LIN {X 0,Y 418.26,Z 256.009,A -85,B 0,C 180,E1 -10305.113,E2 -10305.113} C_VEL
LIN {X 0,Y 418.269,Z 256.008,A -85,B 0,C 180,E1 -10308.419,E2 -10308.419} C_VEL
LIN {X 0,Y 418.275,Z 256.076,A -85,B 0,C 180,E1 -10308.94,E2 -10308.94} C_VEL
LIN {X 0,Y 420.863,Z 267.45,A -85,B 0,C 180,E1 -10311.704,E2 -10311.704} C_VEL
LIN {X 0,Y 421.563,Z 270.846,A -85,B 0,C 180,E1 -10312.505,E2 -10312.505} C_VEL
LIN {X 0,Y 424.681,Z 279.122,A -85,B 0,C 180,E1 -10312.884,E2 -10312.884} C_VEL
LIN {X 0,Y 428.293,Z 295.182,A -85,B 0,C 180,E1 -10313.417,E2 -10313.417} C_VEL
LIN {X 0,Y 426.388,Z 407.598,A -85,B 0,C 180,E1 -10315.38,E2 -10315.38} C_VEL
LIN {X 0,Y 425.814,Z 421.951,A -85,B 0,C 180,E1 -10315.821,E2 -10315.821} C_VEL
LIN {X 0,Y 425.057,Z 435.648,A -85,B 0,C 180,E1 -10316.437,E2 -10316.437} C_VEL
LIN {X 0,Y 424.136,Z 449.482,A -85,B 0,C 180,E1 -10317.277,E2 -10317.277} C_VEL
LIN {X 0,Y 423.118,Z 462.711,A -85,B 0,C 180,E1 -10318.313,E2 -10318.313} C_VEL
LIN {X 0,Y 421.977,Z 474.603,A -85,B 0,C 180,E1 -10319.472,E2 -10319.472} C_VEL
LIN {X 0,Y 420.938,Z 485.519,A -85,B 0,C 180,E1 -10320.784,E2 -10320.784} C_VEL
LIN {X 0,Y 420.063,Z 494.402,A -85,B 0,C 180,E1 -10322.066,E2 -10322.066} C_VEL
LIN {X 0,Y 419.198,Z 503.344,A -85,B 0,C 180,E1 -10323.623,E2 -10323.623} C_VEL
LIN {X 0,Y 418.524,Z 510.7,A -85,B 0,C 180,E1 -10325.178,E2 -10325.178} C_VEL
LIN {X 0,Y 417.991,Z 516.714,A -85,B 0,C 180,E1 -10326.727,E2 -10326.727} C_VEL
LIN {X 0,Y 417.581,Z 521.545,A -85,B 0,C 180,E1 -10328.269,E2 -10328.269} C_VEL
LIN {X 0,Y 417.325,Z 525.36,A -85,B 0,C 180,E1 -10329.805,E2 -10329.805} C_VEL
LIN {X 0,Y 417.115,Z 528.26,A -85,B 0,C 180,E1 -10331.33,E2 -10331.33} C_VEL
LIN {X 0,Y 416.933,Z 530.732,A -85,B 0,C 180,E1 -10333.348,E2 -10333.348} C_VEL
LIN {X 0,Y 416.946,Z 531.423,A -85,B 0,C 180,E1 -10334.354,E2 -10334.354} C_VEL
LIN {X 0,Y 416.871,Z 531.754,A -85,B 0,C 180,E1 -10336.33,E2 -10336.33} C_VEL
LIN {X 0,Y 416.228,Z 531.607,A -85,B 0,C 180,E1 -10337.138,E2 -10337.138} C_VEL
LIN {X 0,Y 413.366,Z 530.788,A -85,B 0,C 180,E1 -10338.446,E2 -10338.446} C_VEL
LIN {X 0,Y 410.965,Z 529.637,A -85,B 0,C 180,E1 -10339.495,E2 -10339.495} C_VEL
LIN {X 0,Y 409.941,Z 528.316,A -85,B 0,C 180,E1 -10340.434,E2 -10340.434} C_VEL
LIN {X 0,Y 409.937,Z 528.026,A -85,B 0,C 180,E1 -10340.57,E2 -10340.57} C_VEL
LIN {X 0,Y 410.167,Z 525.049,A -85,B 0,C 180,E1 -10342.122,E2 -10342.122} C_VEL
LIN {X 0,Y 410.467,Z 519.827,A -85,B 0,C 180,E1 -10344.104,E2 -10344.104} C_VEL
LIN {X 0,Y 410.76,Z 514.771,A -85,B 0,C 180,E1 -10345.584,E2 -10345.584} C_VEL
LIN {X 0,Y 411.274,Z 507.569,A -85,B 0,C 180,E1 -10347.307,E2 -10347.307} C_VEL
LIN {X 0,Y 411.955,Z 500.022,A -85,B 0,C 180,E1 -10348.778,E2 -10348.778} C_VEL
LIN {X 0,Y 412.765,Z 490.981,A -85,B 0,C 180,E1 -10350.244,E2 -10350.244} C_VEL
LIN {X 0,Y 413.718,Z 480.057,A -85,B 0,C 180,E1 -10351.704,E2 -10351.704} C_VEL
LIN {X 0,Y 414.695,Z 468.928,A -85,B 0,C 180,E1 -10352.914,E2 -10352.914} C_VEL
LIN {X 0,Y 415.654,Z 456.533,A -85,B 0,C 180,E1 -10354.009,E2 -10354.009} C_VEL
LIN {X 0,Y 416.492,Z 443.925,A -85,B 0,C 180,E1 -10354.9,E2 -10354.9} C_VEL
LIN {X 0,Y 417.184,Z 430.594,A -85,B 0,C 180,E1 -10355.631,E2 -10355.631} C_VEL
LIN {X 0,Y 417.775,Z 416.637,A -85,B 0,C 180,E1 -10356.187,E2 -10356.187} C_VEL
LIN {X 0,Y 418.145,Z 402.956,A -85,B 0,C 180,E1 -10356.545,E2 -10356.545} C_VEL
LIN {X 0,Y 419.744,Z 296.011,A -85,B 0,C 180,E1 -10358.395,E2 -10358.395} C_VEL
LIN {X 0,Y 416.319,Z 279.208,A -85,B 0,C 180,E1 -10358.869,E2 -10358.869} C_VEL
LIN {X 0,Y 414.122,Z 270.702,A -85,B 0,C 180,E1 -10359.143,E2 -10359.143} C_VEL
LIN {X 0,Y 411.36,Z 256.874,A -85,B 0,C 180,E1 -10362.3,E2 -10362.3} C_VEL
LIN {X 0,Y 411.242,Z 256.887,A -85,B 0,C 180,E1 -10365.869,E2 -10365.869} C_VEL
LIN {X 0,Y 411.222,Z 256.883,A -85,B 0,C 180,E1 -10368.948,E2 -10368.948} C_VEL
LIN {X 0,Y 411.192,Z 256.889,A -85,B 0,C 180,E1 -10372.087,E2 -10372.087} C_VEL
LIN {X 0,Y 411.224,Z 256.885,A -85,B 0,C 180,E1 -10375.293,E2 -10375.293} C_VEL
LIN {X 0,Y 411.21,Z 256.884,A -85,B 0,C 180,E1 -10378.59,E2 -10378.59} C_VEL
LIN {X 0,Y 411.158,Z 256.893,A -85,B 0,C 180,E1 -10381.997,E2 -10381.997} C_VEL
LIN {X 0,Y 411.186,Z 256.894,A -85,B 0,C 180,E1 -10385.529,E2 -10385.529} C_VEL
LIN {X 0,Y 411.219,Z 256.888,A -85,B 0,C 180,E1 -10389.223,E2 -10389.223} C_VEL
LIN {X 0,Y 411.219,Z 256.884,A -85,B 0,C 180,E1 -10392.704,E2 -10392.704} C_VEL
LIN {X 0,Y 411.218,Z 256.884,A -85,B 0,C 180,E1 -10395.873,E2 -10395.873} C_VEL
LIN {X 0,Y 411.197,Z 256.887,A -85,B 0,C 180,E1 -10398.765,E2 -10398.765} C_VEL
LIN {X 0,Y 411.192,Z 256.886,A -85,B 0,C 180,E1 -10402.028,E2 -10402.028} C_VEL
LIN {X 0,Y 411.194,Z 256.887,A -85,B 0,C 180,E1 -10405.667,E2 -10405.667} C_VEL
LIN {X 0,Y 411.186,Z 256.893,A -85,B 0,C 180,E1 -10409.154,E2 -10409.154} C_VEL
LIN {X 0,Y 411.248,Z 256.881,A -85,B 0,C 180,E1 -10412.523,E2 -10412.523} C_VEL
LIN {X 0,Y 411.216,Z 256.883,A -85,B 0,C 180,E1 -10415.786,E2 -10415.786} C_VEL
LIN {X 0,Y 411.185,Z 256.893,A -85,B 0,C 180,E1 -10418.967,E2 -10418.967} C_VEL
LIN {X 0,Y 411.242,Z 256.88,A -85,B 0,C 180,E1 -10422.086,E2 -10422.086} C_VEL
LIN {X 0,Y 411.253,Z 256.881,A -85,B 0,C 180,E1 -10425.149,E2 -10425.149} C_VEL
LIN {X 0,Y 411.275,Z 256.877,A -85,B 0,C 180,E1 -10428.169,E2 -10428.169} C_VEL
LIN {X 0,Y 411.432,Z 256.859,A -85,B 0,C 180,E1 -10432.19,E2 -10432.19} C_VEL
LIN {X 0,Y 411.468,Z 256.854,A -85,B 0,C 180,E1 -10434.119,E2 -10434.119} C_VEL
LIN {X 0,Y 411.506,Z 256.849,A -85,B 0,C 180,E1 -10438.044,E2 -10438.044} C_VEL
LIN {X 0,Y 411.634,Z 256.833,A -85,B 0,C 180,E1 -10440.001,E2 -10440.001} C_VEL
LIN {X 0,Y 411.459,Z 256.855,A -85,B 0,C 180,E1 -10442.939,E2 -10442.939} C_VEL
LIN {X 0,Y 411.45,Z 256.856,A -85,B 0,C 180,E1 -10446.868,E2 -10446.868} C_VEL
LIN {X 0,Y 411.287,Z 256.876,A -85,B 0,C 180,E1 -10449.84,E2 -10449.84} C_VEL
LIN {X 0,Y 411.3,Z 256.873,A -85,B 0,C 180,E1 -10453.105,E2 -10453.105} C_VEL
LIN {X 0,Y 411.259,Z 256.878,A -85,B 0,C 180,E1 -10456.871,E2 -10456.871} C_VEL
LIN {X 0,Y 411.226,Z 256.887,A -85,B 0,C 180,E1 -10459.988,E2 -10459.988} C_VEL
LIN {X 0,Y 411.193,Z 256.886,A -85,B 0,C 180,E1 -10463.149,E2 -10463.149} C_VEL
LIN {X 0,Y 411.235,Z 256.884,A -85,B 0,C 180,E1 -10466.382,E2 -10466.382} C_VEL
LIN {X 0,Y 411.208,Z 256.888,A -85,B 0,C 180,E1 -10469.713,E2 -10469.713} C_VEL
LIN {X 0,Y 411.205,Z 256.885,A -85,B 0,C 180,E1 -10473.157,E2 -10473.157} C_VEL
LIN {X 0,Y 411.194,Z 256.886,A -85,B 0,C 180,E1 -10476.554,E2 -10476.554} C_VEL
LIN {X 0,Y 411.217,Z 256.89,A -85,B 0,C 180,E1 -10479.73,E2 -10479.73} C_VEL
LIN {X 0,Y 411.173,Z 256.89,A -85,B 0,C 180,E1 -10483.135,E2 -10483.135} C_VEL
LIN {X 0,Y 411.168,Z 256.894,A -85,B 0,C 180,E1 -10485.882,E2 -10485.882} C_VEL
LIN {X 0,Y 411.163,Z 256.89,A -85,B 0,C 180,E1 -10488.773,E2 -10488.773} C_VEL
LIN {X 0,Y 411.191,Z 256.888,A -85,B 0,C 180,E1 -10492.027,E2 -10492.027} C_VEL
LIN {X 0,Y 411.207,Z 256.892,A -85,B 0,C 180,E1 -10495.667,E2 -10495.667} C_VEL
LIN {X 0,Y 411.193,Z 256.895,A -85,B 0,C 180,E1 -10499.153,E2 -10499.153} C_VEL
LIN {X 0,Y 411.266,Z 257.003,A -85,B 0,C 180,E1 -10500.187,E2 -10500.187} C_VEL
LIN {X 0,Y 414.273,Z 270.814,A -85,B 0,C 180,E1 -10503.013,E2 -10503.013} C_VEL
LIN {X 0,Y 415.359,Z 276.668,A -85,B 0,C 180,E1 -10504.171,E2 -10504.171} C_VEL
LIN {X 0,Y 414.479,Z 290.188,A -85,B 0,C 180,E1 -10506.632,E2 -10506.632} C_VEL
LIN {X 0,Y 414.348,Z 291.589,A -85,B 0,C 180,E1 -10506.883,E2 -10506.883} C_VEL
LIN {X 0,Y 419.501,Z 322.053,A -85,B 0,C 180,E1 -10507.697,E2 -10507.697} C_VEL
LIN {X 0,Y 417.904,Z 429.765,A -85,B 0,C 180,E1 -10509.577,E2 -10509.577} C_VEL
LIN {X 0,Y 417.294,Z 444.417,A -85,B 0,C 180,E1 -10510.028,E2 -10510.028} C_VEL
LIN {X 0,Y 416.495,Z 458.845,A -85,B 0,C 180,E1 -10510.684,E2 -10510.684} C_VEL
LIN {X 0,Y 415.673,Z 472.379,A -85,B 0,C 180,E1 -10511.518,E2 -10511.518} C_VEL
LIN {X 0,Y 414.678,Z 484.854,A -85,B 0,C 180,E1 -10512.493,E2 -10512.493} C_VEL
LIN {X 0,Y 413.792,Z 496.271,A -85,B 0,C 180,E1 -10513.599,E2 -10513.599} C_VEL
LIN {X 0,Y 412.87,Z 505.762,A -85,B 0,C 180,E1 -10514.702,E2 -10514.702} C_VEL
LIN {X 0,Y 412.026,Z 516.36,A -85,B 0,C 180,E1 -10516.184,E2 -10516.184} C_VEL
LIN {X 0,Y 411.352,Z 525.09,A -85,B 0,C 180,E1 -10517.669,E2 -10517.669} C_VEL
LIN {X 0,Y 410.726,Z 533.442,A -85,B 0,C 180,E1 -10519.401,E2 -10519.401} C_VEL
LIN {X 0,Y 410.337,Z 540.142,A -85,B 0,C 180,E1 -10521.133,E2 -10521.133} C_VEL
LIN {X 0,Y 410.086,Z 546.078,A -85,B 0,C 180,E1 -10523.11,E2 -10523.11} C_VEL
LIN {X 0,Y 409.983,Z 550.415,A -85,B 0,C 180,E1 -10525.083,E2 -10525.083} C_VEL
LIN {X 0,Y 409.916,Z 553.287,A -85,B 0,C 180,E1 -10527.052,E2 -10527.052} C_VEL
LIN {X 0,Y 409.935,Z 554.78,A -85,B 0,C 180,E1 -10529.018,E2 -10529.018} C_VEL
LIN {X 0,Y 409.935,Z 554.928,A -85,B 0,C 180,E1 -10530.982,E2 -10530.982} C_VEL
LIN {X 0,Y 409.912,Z 553.743,A -85,B 0,C 180,E1 -10532.948,E2 -10532.948} C_VEL
LIN {X 0,Y 409.988,Z 551.208,A -85,B 0,C 180,E1 -10534.917,E2 -10534.917} C_VEL
LIN {X 0,Y 410.089,Z 547.236,A -85,B 0,C 180,E1 -10536.89,E2 -10536.89} C_VEL
LIN {X 0,Y 410.397,Z 541.707,A -85,B 0,C 180,E1 -10538.866,E2 -10538.866} C_VEL
LIN {X 0,Y 410.798,Z 535.489,A -85,B 0,C 180,E1 -10540.597,E2 -10540.597} C_VEL
LIN {X 0,Y 411.601,Z 527.762,A -85,B 0,C 180,E1 -10542.323,E2 -10542.323} C_VEL
LIN {X 0,Y 412.242,Z 519.724,A -85,B 0,C 180,E1 -10543.808,E2 -10543.808} C_VEL
LIN {X 0,Y 413.21,Z 510.058,A -85,B 0,C 180,E1 -10545.285,E2 -10545.285} C_VEL
LIN {X 0,Y 414.319,Z 499.36,A -85,B 0,C 180,E1 -10546.633,E2 -10546.633} C_VEL
LIN {X 0,Y 415.581,Z 487.541,A -85,B 0,C 180,E1 -10547.849,E2 -10547.849} C_VEL
LIN {X 0,Y 416.605,Z 475.974,A -85,B 0,C 180,E1 -10548.822,E2 -10548.822} C_VEL
LIN {X 0,Y 417.696,Z 462.417,A -85,B 0,C 180,E1 -10549.728,E2 -10549.728} C_VEL
LIN {X 0,Y 418.592,Z 449.41,A -85,B 0,C 180,E1 -10550.388,E2 -10550.388} C_VEL
LIN {X 0,Y 419.315,Z 435.504,A -85,B 0,C 180,E1 -10550.896,E2 -10550.896} C_VEL
LIN {X 0,Y 419.838,Z 421.043,A -85,B 0,C 180,E1 -10551.222,E2 -10551.222} C_VEL
LIN {X 0,Y 421.421,Z 321.827,A -85,B 0,C 180,E1 -10552.968,E2 -10552.968} C_VEL
LIN {X 0,Y 417.71,Z 302.021,A -85,B 0,C 180,E1 -10553.589,E2 -10553.589} C_VEL
LIN {X 0,Y 415.388,Z 291.087,A -85,B 0,C 180,E1 -10553.986,E2 -10553.986} C_VEL
LIN {X 0,Y 416.384,Z 280.226,A -85,B 0,C 180,E1 -10556.029,E2 -10556.029} C_VEL
LIN {X 0,Y 415.006,Z 272.397,A -85,B 0,C 180,E1 -10557.681,E2 -10557.681} C_VEL
LIN {X 0,Y 411.947,Z 259.825,A -85,B 0,C 180,E1 -10560.499,E2 -10560.499} C_VEL
LIN {X 0,Y 411.187,Z 256.895,A -85,B 0,C 180,E1 -10561.183,E2 -10561.183} C_VEL
LIN {X 0,Y 411.206,Z 256.891,A -85,B 0,C 180,E1 -10564.332,E2 -10564.332} C_VEL
LIN {X 0,Y 411.194,Z 256.888,A -85,B 0,C 180,E1 -10567.973,E2 -10567.973} C_VEL
LIN {X 0,Y 411.204,Z 256.884,A -85,B 0,C 180,E1 -10571.234,E2 -10571.234} C_VEL
LIN {X 0,Y 411.223,Z 256.889,A -85,B 0,C 180,E1 -10574.483,E2 -10574.483} C_VEL
LIN {X 0,Y 411.175,Z 256.892,A -85,B 0,C 180,E1 -10578.193,E2 -10578.193} C_VEL
LIN {X 0,Y 411.216,Z 256.886,A -85,B 0,C 180,E1 -10580.775,E2 -10580.775} C_VEL
LIN {X 0,Y 411.195,Z 256.873,A -85,B 0,C 180,E1 -10584.47,E2 -10584.47} C_VEL
LIN {X 0,Y 411.204,Z 256.886,A -85,B 0,C 180,E1 -10586.872,E2 -10586.872} C_VEL
LIN {X 0,Y 411.236,Z 256.883,A -85,B 0,C 180,E1 -10590.641,E2 -10590.641} C_VEL
LIN {X 0,Y 411.233,Z 256.884,A -85,B 0,C 180,E1 -10593.618,E2 -10593.618} C_VEL
LIN {X 0,Y 411.198,Z 256.885,A -85,B 0,C 180,E1 -10596.851,E2 -10596.851} C_VEL
LIN {X 0,Y 411.209,Z 256.884,A -85,B 0,C 180,E1 -10600.049,E2 -10600.049} C_VEL
LIN {X 0,Y 411.257,Z 256.881,A -85,B 0,C 180,E1 -10603.13,E2 -10603.13} C_VEL
LIN {X 0,Y 411.298,Z 256.875,A -85,B 0,C 180,E1 -10606.895,E2 -10606.895} C_VEL
LIN {X 0,Y 411.286,Z 256.877,A -85,B 0,C 180,E1 -10610.16,E2 -10610.16} C_VEL
LIN {X 0,Y 411.448,Z 256.851,A -85,B 0,C 180,E1 -10613.132,E2 -10613.132} C_VEL
LIN {X 0,Y 411.304,Z 256.877,A -85,B 0,C 180,E1 -10615.098,E2 -10615.098} C_VEL
LIN {X 0,Y 411.505,Z 256.848,A -85,B 0,C 180,E1 -10618.041,E2 -10618.041} C_VEL
LIN {X 0,Y 411.634,Z 256.831,A -85,B 0,C 180,E1 -10619.999,E2 -10619.999} C_VEL
LIN {X 0,Y 411.457,Z 256.856,A -85,B 0,C 180,E1 -10622.936,E2 -10622.936} C_VEL
LIN {X 0,Y 411.446,Z 256.856,A -85,B 0,C 180,E1 -10626.866,E2 -10626.866} C_VEL
LIN {X 0,Y 411.283,Z 256.872,A -85,B 0,C 180,E1 -10629.838,E2 -10629.838} C_VEL
LIN {X 0,Y 411.294,Z 256.874,A -85,B 0,C 180,E1 -10633.103,E2 -10633.103} C_VEL
LIN {X 0,Y 411.246,Z 256.881,A -85,B 0,C 180,E1 -10636.888,E2 -10636.888} C_VEL
LIN {X 0,Y 411.243,Z 256.881,A -85,B 0,C 180,E1 -10639.984,E2 -10639.984} C_VEL
LIN {X 0,Y 411.193,Z 256.887,A -85,B 0,C 180,E1 -10643.146,E2 -10643.146} C_VEL
LIN {X 0,Y 411.225,Z 256.887,A -85,B 0,C 180,E1 -10646.38,E2 -10646.38} C_VEL
LIN {X 0,Y 411.197,Z 256.883,A -85,B 0,C 180,E1 -10649.711,E2 -10649.711} C_VEL
LIN {X 0,Y 411.193,Z 256.89,A -85,B 0,C 180,E1 -10653.155,E2 -10653.155} C_VEL
LIN {X 0,Y 411.182,Z 256.891,A -85,B 0,C 180,E1 -10656.552,E2 -10656.552} C_VEL
LIN {X 0,Y 411.214,Z 256.883,A -85,B 0,C 180,E1 -10659.73,E2 -10659.73} C_VEL
LIN {X 0,Y 411.21,Z 256.889,A -85,B 0,C 180,E1 -10663.126,E2 -10663.126} C_VEL
LIN {X 0,Y 411.225,Z 256.888,A -85,B 0,C 180,E1 -10665.87,E2 -10665.87} C_VEL
LIN {X 0,Y 411.238,Z 256.979,A -85,B 0,C 180,E1 -10668.521,E2 -10668.521} C_VEL
LIN {X 0,Y 413.858,Z 268.368,A -85,B 0,C 180,E1 -10671.364,E2 -10671.364} C_VEL
LIN {X 0,Y 414.478,Z 271.288,A -85,B 0,C 180,E1 -10672.033,E2 -10672.033} C_VEL
LIN {X 0,Y 418.608,Z 281.644,A -85,B 0,C 180,E1 -10672.52,E2 -10672.52} C_VEL
LIN {X 0,Y 421.885,Z 296.394,A -85,B 0,C 180,E1 -10673.02,E2 -10673.02} C_VEL
LIN {X 0,Y 419.885,Z 407.614,A -85,B 0,C 180,E1 -10674.991,E2 -10674.991} C_VEL
LIN {X 0,Y 419.291,Z 422.045,A -85,B 0,C 180,E1 -10675.44,E2 -10675.44} C_VEL
LIN {X 0,Y 418.501,Z 435.628,A -85,B 0,C 180,E1 -10676.057,E2 -10676.057} C_VEL
LIN {X 0,Y 417.602,Z 448.558,A -85,B 0,C 180,E1 -10676.843,E2 -10676.843} C_VEL
LIN {X 0,Y 416.665,Z 460.531,A -85,B 0,C 180,E1 -10677.767,E2 -10677.767} C_VEL
LIN {X 0,Y 415.412,Z 472.812,A -85,B 0,C 180,E1 -10678.936,E2 -10678.936} C_VEL
LIN {X 0,Y 414.428,Z 482.96,A -85,B 0,C 180,E1 -10680.123,E2 -10680.123} C_VEL
LIN {X 0,Y 413.501,Z 491.506,A -85,B 0,C 180,E1 -10681.306,E2 -10681.306} C_VEL
LIN {X 0,Y 412.563,Z 501.016,A -85,B 0,C 180,E1 -10682.892,E2 -10682.892} C_VEL
LIN {X 0,Y 411.752,Z 508.807,A -85,B 0,C 180,E1 -10684.471,E2 -10684.471} C_VEL
LIN {X 0,Y 411.051,Z 516.145,A -85,B 0,C 180,E1 -10686.31,E2 -10686.31} C_VEL
LIN {X 0,Y 410.588,Z 521.136,A -85,B 0,C 180,E1 -10687.879,E2 -10687.879} C_VEL
LIN {X 0,Y 410.296,Z 525.106,A -85,B 0,C 180,E1 -10689.443,E2 -10689.443} C_VEL
LIN {X 0,Y 410.057,Z 528.127,A -85,B 0,C 180,E1 -10690.996,E2 -10690.996} C_VEL
LIN {X 0,Y 409.87,Z 530.765,A -85,B 0,C 180,E1 -10693.053,E2 -10693.053} C_VEL
LIN {X 0,Y 409.794,Z 531.932,A -85,B 0,C 180,E1 -10695.093,E2 -10695.093} C_VEL
LIN {X 0,Y 409.801,Z 531.7,A -85,B 0,C 180,E1 -10697.118,E2 -10697.118} C_VEL
LIN {X 0,Y 409.901,Z 531.063,A -85,B 0,C 180,E1 -10698.127,E2 -10698.127} C_VEL
LIN {X 0,Y 409.891,Z 528.77,A -85,B 0,C 180,E1 -10700.128,E2 -10700.128} C_VEL
LIN {X 0,Y 409.937,Z 528.026,A -85,B 0,C 180,E1 -10700.57,E2 -10700.57} C_VEL
LIN {X 0,Y 409.381,Z 526.68,A -85,B 0,C 180,E1 -10701.368,E2 -10701.368} C_VEL
LIN {X 0,Y 406.708,Z 523.977,A -85,B 0,C 180,E1 -10702.657,E2 -10702.657} C_VEL
LIN {X 0,Y 404.439,Z 521.442,A -85,B 0,C 180,E1 -10703.678,E2 -10703.678} C_VEL
LIN {X 0,Y 403.513,Z 519.237,A -85,B 0,C 180,E1 -10704.45,E2 -10704.45} C_VEL
LIN {X 0,Y 403.466,Z 518.413,A -85,B 0,C 180,E1 -10704.707,E2 -10704.707} C_VEL
LIN {X 0,Y 403.953,Z 511.852,A -85,B 0,C 180,E1 -10706.509,E2 -10706.509} C_VEL
LIN {X 0,Y 404.646,Z 503.899,A -85,B 0,C 180,E1 -10708.258,E2 -10708.258} C_VEL
LIN {X 0,Y 405.387,Z 495.596,A -85,B 0,C 180,E1 -10709.752,E2 -10709.752} C_VEL
LIN {X 0,Y 406.318,Z 485.612,A -85,B 0,C 180,E1 -10711.239,E2 -10711.239} C_VEL
LIN {X 0,Y 407.368,Z 474.474,A -85,B 0,C 180,E1 -10712.596,E2 -10712.596} C_VEL
LIN {X 0,Y 408.416,Z 462.013,A -85,B 0,C 180,E1 -10713.823,E2 -10713.823} C_VEL
LIN {X 0,Y 409.334,Z 449.761,A -85,B 0,C 180,E1 -10714.795,E2 -10714.795} C_VEL
LIN {X 0,Y 410.156,Z 435.959,A -85,B 0,C 180,E1 -10715.654,E2 -10715.654} C_VEL
LIN {X 0,Y 410.805,Z 422.179,A -85,B 0,C 180,E1 -10716.292,E2 -10716.292} C_VEL
LIN {X 0,Y 411.287,Z 407.832,A -85,B 0,C 180,E1 -10716.747,E2 -10716.747} C_VEL
LIN {X 0,Y 413.052,Z 297.138,A -85,B 0,C 180,E1 -10718.708,E2 -10718.708} C_VEL
LIN {X 0,Y 409.248,Z 278.323,A -85,B 0,C 180,E1 -10719.25,E2 -10719.25} C_VEL
LIN {X 0,Y 406.953,Z 270.822,A -85,B 0,C 180,E1 -10719.529,E2 -10719.529} C_VEL
LIN {X 0,Y 404.27,Z 257.755,A -85,B 0,C 180,E1 -10722.583,E2 -10722.583} C_VEL
LIN {X 0,Y 404.208,Z 257.76,A -85,B 0,C 180,E1 -10726.152,E2 -10726.152} C_VEL
LIN {X 0,Y 404.175,Z 257.762,A -85,B 0,C 180,E1 -10729.292,E2 -10729.292} C_VEL
LIN {X 0,Y 404.142,Z 257.764,A -85,B 0,C 180,E1 -10732.835,E2 -10732.835} C_VEL
LIN {X 0,Y 404.171,Z 257.767,A -85,B 0,C 180,E1 -10735.767,E2 -10735.767} C_VEL
LIN {X 0,Y 404.184,Z 257.762,A -85,B 0,C 180,E1 -10738,E2 -10738} C_VEL
LIN {X 0,Y 404.136,Z 257.771,A -85,B 0,C 180,E1 -10741.446,E2 -10741.446} C_VEL
LIN {X 0,Y 404.172,Z 257.763,A -85,B 0,C 180,E1 -10745.017,E2 -10745.017} C_VEL
LIN {X 0,Y 404.151,Z 257.764,A -85,B 0,C 180,E1 -10748.756,E2 -10748.756} C_VEL
LIN {X 0,Y 404.179,Z 257.764,A -85,B 0,C 180,E1 -10751.611,E2 -10751.611} C_VEL
LIN {X 0,Y 404.188,Z 257.759,A -85,B 0,C 180,E1 -10754.531,E2 -10754.531} C_VEL
LIN {X 0,Y 404.194,Z 257.765,A -85,B 0,C 180,E1 -10757.306,E2 -10757.306} C_VEL
LIN {X 0,Y 404.156,Z 257.763,A -85,B 0,C 180,E1 -10759.956,E2 -10759.956} C_VEL
LIN {X 0,Y 404.129,Z 257.773,A -85,B 0,C 180,E1 -10763.125,E2 -10763.125} C_VEL
LIN {X 0,Y 404.133,Z 257.766,A -85,B 0,C 180,E1 -10766.189,E2 -10766.189} C_VEL
LIN {X 0,Y 404.142,Z 257.765,A -85,B 0,C 180,E1 -10769.717,E2 -10769.717} C_VEL
LIN {X 0,Y 404.184,Z 257.764,A -85,B 0,C 180,E1 -10773.124,E2 -10773.124} C_VEL
LIN {X 0,Y 404.166,Z 257.764,A -85,B 0,C 180,E1 -10775.335,E2 -10775.335} C_VEL
LIN {X 0,Y 404.128,Z 257.77,A -85,B 0,C 180,E1 -10778.582,E2 -10778.582} C_VEL
LIN {X 0,Y 404.2,Z 257.757,A -85,B 0,C 180,E1 -10781.763,E2 -10781.763} C_VEL
LIN {X 0,Y 404.198,Z 257.763,A -85,B 0,C 180,E1 -10784.883,E2 -10784.883} C_VEL
LIN {X 0,Y 404.247,Z 257.752,A -85,B 0,C 180,E1 -10787.96,E2 -10787.96} C_VEL
LIN {X 0,Y 404.397,Z 257.734,A -85,B 0,C 180,E1 -10792.13,E2 -10792.13} C_VEL
LIN {X 0,Y 404.416,Z 257.731,A -85,B 0,C 180,E1 -10794.016,E2 -10794.016} C_VEL
LIN {X 0,Y 404.475,Z 257.725,A -85,B 0,C 180,E1 -10798.01,E2 -10798.01} C_VEL
LIN {X 0,Y 404.604,Z 257.709,A -85,B 0,C 180,E1 -10800.001,E2 -10800.001} C_VEL
LIN {X 0,Y 404.416,Z 257.732,A -85,B 0,C 180,E1 -10802.99,E2 -10802.99} C_VEL
LIN {X 0,Y 404.396,Z 257.734,A -85,B 0,C 180,E1 -10806.989,E2 -10806.989} C_VEL
LIN {X 0,Y 404.252,Z 257.754,A -85,B 0,C 180,E1 -10810.013,E2 -10810.013} C_VEL
LIN {X 0,Y 404.261,Z 257.749,A -85,B 0,C 180,E1 -10813.213,E2 -10813.213} C_VEL
LIN {X 0,Y 404.214,Z 257.756,A -85,B 0,C 180,E1 -10817.01,E2 -10817.01} C_VEL
LIN {X 0,Y 404.16,Z 257.766,A -85,B 0,C 180,E1 -10820.353,E2 -10820.353} C_VEL
LIN {X 0,Y 404.16,Z 257.764,A -85,B 0,C 180,E1 -10823.576,E2 -10823.576} C_VEL
LIN {X 0,Y 404.18,Z 257.764,A -85,B 0,C 180,E1 -10825.768,E2 -10825.768} C_VEL
LIN {X 0,Y 404.195,Z 257.765,A -85,B 0,C 180,E1 -10828.001,E2 -10828.001} C_VEL
LIN {X 0,Y 404.143,Z 257.767,A -85,B 0,C 180,E1 -10831.561,E2 -10831.561} C_VEL
LIN {X 0,Y 404.184,Z 257.759,A -85,B 0,C 180,E1 -10835.017,E2 -10835.017} C_VEL
LIN {X 0,Y 404.158,Z 257.762,A -85,B 0,C 180,E1 -10838.758,E2 -10838.758} C_VEL
LIN {X 0,Y 404.123,Z 257.772,A -85,B 0,C 180,E1 -10841.601,E2 -10841.601} C_VEL
LIN {X 0,Y 404.145,Z 257.764,A -85,B 0,C 180,E1 -10844.523,E2 -10844.523} C_VEL
LIN {X 0,Y 404.136,Z 257.768,A -85,B 0,C 180,E1 -10847.297,E2 -10847.297} C_VEL
LIN {X 0,Y 404.17,Z 257.764,A -85,B 0,C 180,E1 -10849.956,E2 -10849.956} C_VEL
LIN {X 0,Y 404.136,Z 257.768,A -85,B 0,C 180,E1 -10853.126,E2 -10853.126} C_VEL
LIN {X 0,Y 404.147,Z 257.769,A -85,B 0,C 180,E1 -10856.189,E2 -10856.189} C_VEL
LIN {X 0,Y 404.199,Z 257.876,A -85,B 0,C 180,E1 -10859.897,E2 -10859.897} C_VEL
LIN {X 0,Y 407.552,Z 273.2,A -85,B 0,C 180,E1 -10863.086,E2 -10863.086} C_VEL
LIN {X 0,Y 408.429,Z 277.816,A -85,B 0,C 180,E1 -10864.016,E2 -10864.016} C_VEL
LIN {X 0,Y 407.533,Z 291.06,A -85,B 0,C 180,E1 -10866.467,E2 -10866.467} C_VEL
LIN {X 0,Y 407.495,Z 291.389,A -85,B 0,C 180,E1 -10866.527,E2 -10866.527} C_VEL
LIN {X 0,Y 412.8,Z 322.934,A -85,B 0,C 180,E1 -10867.386,E2 -10867.386} C_VEL
LIN {X 0,Y 411.173,Z 428.909,A -85,B 0,C 180,E1 -10869.26,E2 -10869.26} C_VEL
LIN {X 0,Y 410.642,Z 443.061,A -85,B 0,C 180,E1 -10869.69,E2 -10869.69} C_VEL
LIN {X 0,Y 409.785,Z 456.796,A -85,B 0,C 180,E1 -10870.299,E2 -10870.299} C_VEL
LIN {X 0,Y 409.034,Z 469.721,A -85,B 0,C 180,E1 -10871.077,E2 -10871.077} C_VEL
LIN {X 0,Y 407.971,Z 482.666,A -85,B 0,C 180,E1 -10872.066,E2 -10872.066} C_VEL
LIN {X 0,Y 406.947,Z 494.426,A -85,B 0,C 180,E1 -10873.186,E2 -10873.186} C_VEL
LIN {X 0,Y 405.942,Z 505.186,A -85,B 0,C 180,E1 -10874.434,E2 -10874.434} C_VEL
LIN {X 0,Y 405.054,Z 515.852,A -85,B 0,C 180,E1 -10875.942,E2 -10875.942} C_VEL
LIN {X 0,Y 404.377,Z 524.644,A -85,B 0,C 180,E1 -10877.453,E2 -10877.453} C_VEL
LIN {X 0,Y 403.686,Z 533.057,A -85,B 0,C 180,E1 -10879.213,E2 -10879.213} C_VEL
LIN {X 0,Y 403.284,Z 539.805,A -85,B 0,C 180,E1 -10880.976,E2 -10880.976} C_VEL
LIN {X 0,Y 403.007,Z 545.776,A -85,B 0,C 180,E1 -10882.988,E2 -10882.988} C_VEL
LIN {X 0,Y 402.895,Z 550.143,A -85,B 0,C 180,E1 -10884.996,E2 -10884.996} C_VEL
LIN {X 0,Y 402.815,Z 553.042,A -85,B 0,C 180,E1 -10887,E2 -10887} C_VEL
LIN {X 0,Y 402.862,Z 554.562,A -85,B 0,C 180,E1 -10889,E2 -10889} C_VEL
LIN {X 0,Y 402.862,Z 554.735,A -85,B 0,C 180,E1 -10890.999,E2 -10890.999} C_VEL
LIN {X 0,Y 402.81,Z 553.574,A -85,B 0,C 180,E1 -10893,E2 -10893} C_VEL
LIN {X 0,Y 402.901,Z 551.068,A -85,B 0,C 180,E1 -10895.003,E2 -10895.003} C_VEL
LIN {X 0,Y 403.033,Z 547.14,A -85,B 0,C 180,E1 -10897.011,E2 -10897.011} C_VEL
LIN {X 0,Y 403.337,Z 541.651,A -85,B 0,C 180,E1 -10899.022,E2 -10899.022} C_VEL
LIN {X 0,Y 403.786,Z 535.472,A -85,B 0,C 180,E1 -10900.784,E2 -10900.784} C_VEL
LIN {X 0,Y 404.625,Z 527.787,A -85,B 0,C 180,E1 -10902.539,E2 -10902.539} C_VEL
LIN {X 0,Y 405.319,Z 519.795,A -85,B 0,C 180,E1 -10904.049,E2 -10904.049} C_VEL
LIN {X 0,Y 406.339,Z 510.183,A -85,B 0,C 180,E1 -10905.55,E2 -10905.55} C_VEL
LIN {X 0,Y 407.538,Z 499.549,A -85,B 0,C 180,E1 -10906.918,E2 -10906.918} C_VEL
LIN {X 0,Y 408.828,Z 487.82,A -85,B 0,C 180,E1 -10908.154,E2 -10908.154} C_VEL
LIN {X 0,Y 409.989,Z 475.02,A -85,B 0,C 180,E1 -10909.25,E2 -10909.25} C_VEL
LIN {X 0,Y 411.144,Z 462.008,A -85,B 0,C 180,E1 -10910.121,E2 -10910.121} C_VEL
LIN {X 0,Y 412.086,Z 448.953,A -85,B 0,C 180,E1 -10910.79,E2 -10910.79} C_VEL
LIN {X 0,Y 412.841,Z 434.911,A -85,B 0,C 180,E1 -10911.305,E2 -10911.305} C_VEL
LIN {X 0,Y 413.359,Z 420.249,A -85,B 0,C 180,E1 -10911.637,E2 -10911.637} C_VEL
LIN {X 0,Y 415.067,Z 323.142,A -85,B 0,C 180,E1 -10913.367,E2 -10913.367} C_VEL
LIN {X 0,Y 411.517,Z 303.949,A -85,B 0,C 180,E1 -10913.98,E2 -10913.98} C_VEL
LIN {X 0,Y 408.681,Z 290.939,A -85,B 0,C 180,E1 -10914.457,E2 -10914.457} C_VEL
LIN {X 0,Y 409.581,Z 281.72,A -85,B 0,C 180,E1 -10916.221,E2 -10916.221} C_VEL
LIN {X 0,Y 407.612,Z 271.555,A -85,B 0,C 180,E1 -10918.436,E2 -10918.436} C_VEL
LIN {X 0,Y 404.126,Z 257.781,A -85,B 0,C 180,E1 -10921.644,E2 -10921.644} C_VEL
LIN {X 0,Y 404.185,Z 257.765,A -85,B 0,C 180,E1 -10925.015,E2 -10925.015} C_VEL
LIN {X 0,Y 404.154,Z 257.774,A -85,B 0,C 180,E1 -10928.756,E2 -10928.756} C_VEL
LIN {X 0,Y 404.187,Z 257.759,A -85,B 0,C 180,E1 -10931.609,E2 -10931.609} C_VEL
LIN {X 0,Y 404.188,Z 257.765,A -85,B 0,C 180,E1 -10934.527,E2 -10934.527} C_VEL
LIN {X 0,Y 404.135,Z 257.767,A -85,B 0,C 180,E1 -10937.294,E2 -10937.294} C_VEL
LIN {X 0,Y 404.167,Z 257.765,A -85,B 0,C 180,E1 -10939.954,E2 -10939.954} C_VEL
LIN {X 0,Y 404.134,Z 257.761,A -85,B 0,C 180,E1 -10943.124,E2 -10943.124} C_VEL
LIN {X 0,Y 404.142,Z 257.764,A -85,B 0,C 180,E1 -10946.186,E2 -10946.186} C_VEL
LIN {X 0,Y 404.149,Z 257.763,A -85,B 0,C 180,E1 -10949.714,E2 -10949.714} C_VEL
LIN {X 0,Y 404.191,Z 257.757,A -85,B 0,C 180,E1 -10953.121,E2 -10953.121} C_VEL
LIN {X 0,Y 404.173,Z 257.764,A -85,B 0,C 180,E1 -10955.333,E2 -10955.333} C_VEL
LIN {X 0,Y 404.133,Z 257.766,A -85,B 0,C 180,E1 -10958.579,E2 -10958.579} C_VEL
LIN {X 0,Y 404.204,Z 257.764,A -85,B 0,C 180,E1 -10961.761,E2 -10961.761} C_VEL
LIN {X 0,Y 404.199,Z 257.755,A -85,B 0,C 180,E1 -10964.881,E2 -10964.881} C_VEL
LIN {X 0,Y 404.25,Z 257.747,A -85,B 0,C 180,E1 -10967.957,E2 -10967.957} C_VEL
LIN {X 0,Y 404.397,Z 257.728,A -85,B 0,C 180,E1 -10972.127,E2 -10972.127} C_VEL
LIN {X 0,Y 404.415,Z 257.733,A -85,B 0,C 180,E1 -10974.014,E2 -10974.014} C_VEL
LIN {X 0,Y 404.474,Z 257.724,A -85,B 0,C 180,E1 -10978.007,E2 -10978.007} C_VEL
LIN {X 0,Y 404.604,Z 257.707,A -85,B 0,C 180,E1 -10979.999,E2 -10979.999} C_VEL
LIN {X 0,Y 404.414,Z 257.734,A -85,B 0,C 180,E1 -10982.987,E2 -10982.987} C_VEL
LIN {X 0,Y 404.393,Z 257.736,A -85,B 0,C 180,E1 -10986.986,E2 -10986.986} C_VEL
LIN {X 0,Y 404.248,Z 257.747,A -85,B 0,C 180,E1 -10990.01,E2 -10990.01} C_VEL
LIN {X 0,Y 404.255,Z 257.749,A -85,B 0,C 180,E1 -10993.21,E2 -10993.21} C_VEL
LIN {X 0,Y 404.204,Z 257.757,A -85,B 0,C 180,E1 -10997.006,E2 -10997.006} C_VEL
LIN {X 0,Y 404.189,Z 257.761,A -85,B 0,C 180,E1 -11000.349,E2 -11000.349} C_VEL
LIN {X 0,Y 404.158,Z 257.761,A -85,B 0,C 180,E1 -11003.573,E2 -11003.573} C_VEL
LIN {X 0,Y 404.182,Z 257.762,A -85,B 0,C 180,E1 -11006.876,E2 -11006.876} C_VEL
LIN {X 0,Y 404.14,Z 257.758,A -85,B 0,C 180,E1 -11010.284,E2 -11010.284} C_VEL
LIN {X 0,Y 404.131,Z 257.769,A -85,B 0,C 180,E1 -11013.811,E2 -11013.811} C_VEL
LIN {X 0,Y 404.127,Z 257.773,A -85,B 0,C 180,E1 -11016.875,E2 -11016.875} C_VEL
LIN {X 0,Y 404.153,Z 257.765,A -85,B 0,C 180,E1 -11020.083,E2 -11020.083} C_VEL
LIN {X 0,Y 404.185,Z 257.764,A -85,B 0,C 180,E1 -11023.09,E2 -11023.09} C_VEL
LIN {X 0,Y 404.198,Z 257.764,A -85,B 0,C 180,E1 -11025.934,E2 -11025.934} C_VEL
LIN {X 0,Y 404.209,Z 257.898,A -85,B 0,C 180,E1 -11028.09,E2 -11028.09} C_VEL
LIN {X 0,Y 406.858,Z 269.347,A -85,B 0,C 180,E1 -11031.013,E2 -11031.013} C_VEL
LIN {X 0,Y 407.285,Z 271.393,A -85,B 0,C 180,E1 -11031.509,E2 -11031.509} C_VEL
LIN {X 0,Y 412.555,Z 284.073,A -85,B 0,C 180,E1 -11032.142,E2 -11032.142} C_VEL
LIN {X 0,Y 415.434,Z 296.833,A -85,B 0,C 180,E1 -11032.59,E2 -11032.59} C_VEL
LIN {X 0,Y 413.442,Z 407.402,A -85,B 0,C 180,E1 -11034.582,E2 -11034.582} C_VEL
LIN {X 0,Y 412.839,Z 421.729,A -85,B 0,C 180,E1 -11035.027,E2 -11035.027} C_VEL
LIN {X 0,Y 411.97,Z 435.745,A -85,B 0,C 180,E1 -11035.668,E2 -11035.668} C_VEL
LIN {X 0,Y 410.957,Z 449.598,A -85,B 0,C 180,E1 -11036.529,E2 -11036.529} C_VEL
LIN {X 0,Y 409.874,Z 462.205,A -85,B 0,C 180,E1 -11037.537,E2 -11037.537} C_VEL
LIN {X 0,Y 408.657,Z 473.537,A -85,B 0,C 180,E1 -11038.653,E2 -11038.653} C_VEL
LIN {X 0,Y 407.498,Z 484.615,A -85,B 0,C 180,E1 -11039.991,E2 -11039.991} C_VEL
LIN {X 0,Y 406.491,Z 493.713,A -85,B 0,C 180,E1 -11041.318,E2 -11041.318} C_VEL
LIN {X 0,Y 405.481,Z 502.933,A -85,B 0,C 180,E1 -11042.937,E2 -11042.937} C_VEL
LIN {X 0,Y 404.681,Z 510.49,A -85,B 0,C 180,E1 -11044.56,E2 -11044.56} C_VEL
LIN {X 0,Y 403.945,Z 517.46,A -85,B 0,C 180,E1 -11046.412,E2 -11046.412} C_VEL
LIN {X 0,Y 403.486,Z 522.232,A -85,B 0,C 180,E1 -11048.008,E2 -11048.008} C_VEL
LIN {X 0,Y 403.182,Z 525.973,A -85,B 0,C 180,E1 -11049.597,E2 -11049.597} C_VEL
LIN {X 0,Y 403.039,Z 527.96,A -85,B 0,C 180,E1 -11050.652,E2 -11050.652} C_VEL
LIN {X 0,Y 402.801,Z 530.768,A -85,B 0,C 180,E1 -11052.746,E2 -11052.746} C_VEL
LIN {X 0,Y 402.721,Z 532.099,A -85,B 0,C 180,E1 -11054.825,E2 -11054.825} C_VEL
LIN {X 0,Y 402.697,Z 532,A -85,B 0,C 180,E1 -11056.887,E2 -11056.887} C_VEL
LIN {X 0,Y 402.8,Z 531.428,A -85,B 0,C 180,E1 -11057.915,E2 -11057.915} C_VEL
LIN {X 0,Y 402.79,Z 529.265,A -85,B 0,C 180,E1 -11059.952,E2 -11059.952} C_VEL
LIN {X 0,Y 403.075,Z 525.677,A -85,B 0,C 180,E1 -11061.982,E2 -11061.982} C_VEL
LIN {X 0,Y 403.357,Z 520.599,A -85,B 0,C 180,E1 -11063.999,E2 -11063.999} C_VEL
LIN {X 0,Y 403.466,Z 518.413,A -85,B 0,C 180,E1 -11064.707,E2 -11064.707} C_VEL
LIN {X 0,Y 402.938,Z 515.927,A -85,B 0,C 180,E1 -11065.466,E2 -11065.466} C_VEL
LIN {X 0,Y 400.424,Z 511.578,A -85,B 0,C 180,E1 -11066.688,E2 -11066.688} C_VEL
LIN {X 0,Y 398.037,Z 506.688,A -85,B 0,C 180,E1 -11067.878,E2 -11067.878} C_VEL
LIN {X 0,Y 397.708,Z 503.341,A -85,B 0,C 180,E1 -11068.579,E2 -11068.579} C_VEL
LIN {X 0,Y 398.615,Z 493.927,A -85,B 0,C 180,E1 -11070.253,E2 -11070.253} C_VEL
LIN {X 0,Y 399.591,Z 483.511,A -85,B 0,C 180,E1 -11071.764,E2 -11071.764} C_VEL
LIN {X 0,Y 400.717,Z 471.853,A -85,B 0,C 180,E1 -11073.142,E2 -11073.142} C_VEL
LIN {X 0,Y 401.726,Z 460.43,A -85,B 0,C 180,E1 -11074.242,E2 -11074.242} C_VEL
LIN {X 0,Y 402.603,Z 448.869,A -85,B 0,C 180,E1 -11075.15,E2 -11075.15} C_VEL
LIN {X 0,Y 403.425,Z 435.164,A -85,B 0,C 180,E1 -11076,E2 -11076} C_VEL
LIN {X 0,Y 404.117,Z 421.01,A -85,B 0,C 180,E1 -11076.647,E2 -11076.647} C_VEL
LIN {X 0,Y 404.583,Z 407.011,A -85,B 0,C 180,E1 -11077.078,E2 -11077.078} C_VEL
LIN {X 0,Y 406.322,Z 297.087,A -85,B 0,C 180,E1 -11079.054,E2 -11079.054} C_VEL
LIN {X 0,Y 402.082,Z 277.658,A -85,B 0,C 180,E1 -11079.643,E2 -11079.643} C_VEL
LIN {X 0,Y 399.729,Z 271.046,A -85,B 0,C 180,E1 -11079.912,E2 -11079.912} C_VEL
LIN {X 0,Y 397.233,Z 258.63,A -85,B 0,C 180,E1 -11082.857,E2 -11082.857} C_VEL
LIN {X 0,Y 397.153,Z 258.636,A -85,B 0,C 180,E1 -11086.447,E2 -11086.447} C_VEL
LIN {X 0,Y 397.152,Z 258.641,A -85,B 0,C 180,E1 -11089.647,E2 -11089.647} C_VEL
LIN {X 0,Y 397.122,Z 258.64,A -85,B 0,C 180,E1 -11093.041,E2 -11093.041} C_VEL
LIN {X 0,Y 397.122,Z 258.64,A -85,B 0,C 180,E1 -11096.259,E2 -11096.259} C_VEL
LIN {X 0,Y 397.113,Z 258.64,A -85,B 0,C 180,E1 -11098.544,E2 -11098.544} C_VEL
LIN {X 0,Y 397.074,Z 258.648,A -85,B 0,C 180,E1 -11101.839,E2 -11101.839} C_VEL
LIN {X 0,Y 397.112,Z 258.64,A -85,B 0,C 180,E1 -11104.494,E2 -11104.494} C_VEL
LIN {X 0,Y 397.097,Z 258.642,A -85,B 0,C 180,E1 -11108.275,E2 -11108.275} C_VEL
LIN {X 0,Y 397.144,Z 258.637,A -85,B 0,C 180,E1 -11111.994,E2 -11111.994} C_VEL
LIN {X 0,Y 397.137,Z 258.641,A -85,B 0,C 180,E1 -11115.06,E2 -11115.06} C_VEL
LIN {X 0,Y 397.143,Z 258.637,A -85,B 0,C 180,E1 -11118.008,E2 -11118.008} C_VEL
LIN {X 0,Y 397.098,Z 258.643,A -85,B 0,C 180,E1 -11121.727,E2 -11121.727} C_VEL
LIN {X 0,Y 397.114,Z 258.643,A -85,B 0,C 180,E1 -11125.508,E2 -11125.508} C_VEL
LIN {X 0,Y 397.073,Z 258.651,A -85,B 0,C 180,E1 -11129.119,E2 -11129.119} C_VEL
LIN {X 0,Y 397.183,Z 258.634,A -85,B 0,C 180,E1 -11132.611,E2 -11132.611} C_VEL
LIN {X 0,Y 397.122,Z 258.639,A -85,B 0,C 180,E1 -11135.983,E2 -11135.983} C_VEL
LIN {X 0,Y 397.128,Z 258.638,A -85,B 0,C 180,E1 -11139.706,E2 -11139.706} C_VEL
LIN {X 0,Y 397.172,Z 258.639,A -85,B 0,C 180,E1 -11142.846,E2 -11142.846} C_VEL
LIN {X 0,Y 397.217,Z 258.633,A -85,B 0,C 180,E1 -11146.68,E2 -11146.68} C_VEL
LIN {X 0,Y 397.209,Z 258.628,A -85,B 0,C 180,E1 -11149.81,E2 -11149.81} C_VEL
LIN {X 0,Y 397.345,Z 258.615,A -85,B 0,C 180,E1 -11152.889,E2 -11152.889} C_VEL
LIN {X 0,Y 397.249,Z 258.626,A -85,B 0,C 180,E1 -11154.927,E2 -11154.927} C_VEL
LIN {X 0,Y 397.444,Z 258.6,A -85,B 0,C 180,E1 -11157.975,E2 -11157.975} C_VEL
LIN {X 0,Y 397.573,Z 258.585,A -85,B 0,C 180,E1 -11160.001,E2 -11160.001} C_VEL
LIN {X 0,Y 397.375,Z 258.608,A -85,B 0,C 180,E1 -11163.043,E2 -11163.043} C_VEL
LIN {X 0,Y 397.367,Z 258.612,A -85,B 0,C 180,E1 -11166.093,E2 -11166.093} C_VEL
LIN {X 0,Y 397.247,Z 258.623,A -85,B 0,C 180,E1 -11169.163,E2 -11169.163} C_VEL
LIN {X 0,Y 397.214,Z 258.635,A -85,B 0,C 180,E1 -11172.26,E2 -11172.26} C_VEL
LIN {X 0,Y 397.179,Z 258.632,A -85,B 0,C 180,E1 -11175.393,E2 -11175.393} C_VEL
LIN {X 0,Y 397.158,Z 258.637,A -85,B 0,C 180,E1 -11178.575,E2 -11178.575} C_VEL
LIN {X 0,Y 397.092,Z 258.646,A -85,B 0,C 180,E1 -11181.82,E2 -11181.82} C_VEL
LIN {X 0,Y 397.15,Z 258.637,A -85,B 0,C 180,E1 -11185.514,E2 -11185.514} C_VEL
LIN {X 0,Y 397.124,Z 258.64,A -85,B 0,C 180,E1 -11188.545,E2 -11188.545} C_VEL
LIN {X 0,Y 397.109,Z 258.645,A -85,B 0,C 180,E1 -11192.07,E2 -11192.07} C_VEL
LIN {X 0,Y 397.118,Z 258.642,A -85,B 0,C 180,E1 -11195.505,E2 -11195.505} C_VEL
LIN {X 0,Y 397.133,Z 258.638,A -85,B 0,C 180,E1 -11198.863,E2 -11198.863} C_VEL
LIN {X 0,Y 397.068,Z 258.647,A -85,B 0,C 180,E1 -11202.268,E2 -11202.268} C_VEL
LIN {X 0,Y 397.087,Z 258.644,A -85,B 0,C 180,E1 -11205.07,E2 -11205.07} C_VEL
LIN {X 0,Y 397.066,Z 258.648,A -85,B 0,C 180,E1 -11208.022,E2 -11208.022} C_VEL
LIN {X 0,Y 397.126,Z 258.641,A -85,B 0,C 180,E1 -11211.141,E2 -11211.141} C_VEL
LIN {X 0,Y 397.12,Z 258.639,A -85,B 0,C 180,E1 -11214.498,E2 -11214.498} C_VEL
LIN {X 0,Y 397.081,Z 258.655,A -85,B 0,C 180,E1 -11217.929,E2 -11217.929} C_VEL
LIN {X 0,Y 397.134,Z 258.659,A -85,B 0,C 180,E1 -11219.576,E2 -11219.576} C_VEL
LIN {X 0,Y 400.226,Z 272.642,A -85,B 0,C 180,E1 -11222.552,E2 -11222.552} C_VEL
LIN {X 0,Y 401.515,Z 279.971,A -85,B 0,C 180,E1 -11224.05,E2 -11224.05} C_VEL
LIN {X 0,Y 400.652,Z 291.232,A -85,B 0,C 180,E1 -11226.168,E2 -11226.168} C_VEL
LIN {X 0,Y 406.097,Z 323.054,A -85,B 0,C 180,E1 -11227.053,E2 -11227.053} C_VEL
LIN {X 0,Y 404.427,Z 429.247,A -85,B 0,C 180,E1 -11228.964,E2 -11228.964} C_VEL
LIN {X 0,Y 403.782,Z 443.952,A -85,B 0,C 180,E1 -11229.429,E2 -11229.429} C_VEL
LIN {X 0,Y 402.951,Z 457.431,A -85,B 0,C 180,E1 -11230.051,E2 -11230.051} C_VEL
LIN {X 0,Y 402.073,Z 471.28,A -85,B 0,C 180,E1 -11230.918,E2 -11230.918} C_VEL
LIN {X 0,Y 401.034,Z 483.357,A -85,B 0,C 180,E1 -11231.877,E2 -11231.877} C_VEL
LIN {X 0,Y 399.978,Z 494.96,A -85,B 0,C 180,E1 -11233.016,E2 -11233.016} C_VEL
LIN {X 0,Y 398.868,Z 506.585,A -85,B 0,C 180,E1 -11234.413,E2 -11234.413} C_VEL
LIN {X 0,Y 397.974,Z 516.867,A -85,B 0,C 180,E1 -11235.931,E2 -11235.931} C_VEL
LIN {X 0,Y 397.254,Z 525.529,A -85,B 0,C 180,E1 -11237.484,E2 -11237.484} C_VEL
LIN {X 0,Y 396.594,Z 533.694,A -85,B 0,C 180,E1 -11239.277,E2 -11239.277} C_VEL
LIN {X 0,Y 396.223,Z 539.446,A -85,B 0,C 180,E1 -11240.814,E2 -11240.814} C_VEL
LIN {X 0,Y 395.928,Z 545.459,A -85,B 0,C 180,E1 -11242.862,E2 -11242.862} C_VEL
LIN {X 0,Y 395.793,Z 549.859,A -85,B 0,C 180,E1 -11244.906,E2 -11244.906} C_VEL
LIN {X 0,Y 395.718,Z 552.79,A -85,B 0,C 180,E1 -11246.946,E2 -11246.946} C_VEL
LIN {X 0,Y 395.791,Z 554.341,A -85,B 0,C 180,E1 -11248.982,E2 -11248.982} C_VEL
LIN {X 0,Y 395.791,Z 554.543,A -85,B 0,C 180,E1 -11251.017,E2 -11251.017} C_VEL
LIN {X 0,Y 395.714,Z 553.41,A -85,B 0,C 180,E1 -11253.054,E2 -11253.054} C_VEL
LIN {X 0,Y 395.8,Z 550.934,A -85,B 0,C 180,E1 -11255.093,E2 -11255.093} C_VEL
LIN {X 0,Y 395.947,Z 547.046,A -85,B 0,C 180,E1 -11257.137,E2 -11257.137} C_VEL
LIN {X 0,Y 396.292,Z 541.598,A -85,B 0,C 180,E1 -11259.184,E2 -11259.184} C_VEL
LIN {X 0,Y 396.679,Z 536.431,A -85,B 0,C 180,E1 -11260.721,E2 -11260.721} C_VEL
LIN {X 0,Y 397.542,Z 529.035,A -85,B 0,C 180,E1 -11262.507,E2 -11262.507} C_VEL
LIN {X 0,Y 398.256,Z 521.222,A -85,B 0,C 180,E1 -11264.061,E2 -11264.061} C_VEL
LIN {X 0,Y 399.291,Z 512.084,A -85,B 0,C 180,E1 -11265.57,E2 -11265.57} C_VEL
LIN {X 0,Y 400.471,Z 501.903,A -85,B 0,C 180,E1 -11266.963,E2 -11266.963} C_VEL
LIN {X 0,Y 401.78,Z 490.724,A -85,B 0,C 180,E1 -11268.22,E2 -11268.22} C_VEL
LIN {X 0,Y 403.058,Z 478.405,A -85,B 0,C 180,E1 -11269.347,E2 -11269.347} C_VEL
LIN {X 0,Y 404.27,Z 465.961,A -85,B 0,C 180,E1 -11270.254,E2 -11270.254} C_VEL
LIN {X 0,Y 405.215,Z 453.7,A -85,B 0,C 180,E1 -11270.959,E2 -11270.959} C_VEL
LIN {X 0,Y 406.155,Z 439.937,A -85,B 0,C 180,E1 -11271.54,E2 -11271.54} C_VEL
LIN {X 0,Y 406.773,Z 425.797,A -85,B 0,C 180,E1 -11271.939,E2 -11271.939} C_VEL
LIN {X 0,Y 408.668,Z 323.789,A -85,B 0,C 180,E1 -11273.796,E2 -11273.796} C_VEL
LIN {X 0,Y 405.197,Z 305.16,A -85,B 0,C 180,E1 -11274.412,E2 -11274.412} C_VEL
LIN {X 0,Y 402.03,Z 290.701,A -85,B 0,C 180,E1 -11274.961,E2 -11274.961} C_VEL
LIN {X 0,Y 402.779,Z 283.247,A -85,B 0,C 180,E1 -11276.419,E2 -11276.419} C_VEL
LIN {X 0,Y 400.688,Z 272.944,A -85,B 0,C 180,E1 -11278.717,E2 -11278.717} C_VEL
LIN {X 0,Y 397.828,Z 261.597,A -85,B 0,C 180,E1 -11281.408,E2 -11281.408} C_VEL
LIN {X 0,Y 397.091,Z 258.648,A -85,B 0,C 180,E1 -11282.144,E2 -11282.144} C_VEL
LIN {X 0,Y 397.12,Z 258.649,A -85,B 0,C 180,E1 -11285.502,E2 -11285.502} C_VEL
LIN {X 0,Y 397.129,Z 258.648,A -85,B 0,C 180,E1 -11288.86,E2 -11288.86} C_VEL
LIN {X 0,Y 397.157,Z 258.64,A -85,B 0,C 180,E1 -11292.254,E2 -11292.254} C_VEL
LIN {X 0,Y 397.109,Z 258.643,A -85,B 0,C 180,E1 -11295.064,E2 -11295.064} C_VEL
LIN {X 0,Y 397.064,Z 258.649,A -85,B 0,C 180,E1 -11298.02,E2 -11298.02} C_VEL
LIN {X 0,Y 397.128,Z 258.64,A -85,B 0,C 180,E1 -11301.137,E2 -11301.137} C_VEL
LIN {X 0,Y 397.116,Z 258.625,A -85,B 0,C 180,E1 -11304.495,E2 -11304.495} C_VEL
LIN {X 0,Y 397.077,Z 258.648,A -85,B 0,C 180,E1 -11307.927,E2 -11307.927} C_VEL
LIN {X 0,Y 397.123,Z 258.642,A -85,B 0,C 180,E1 -11311.455,E2 -11311.455} C_VEL
LIN {X 0,Y 397.148,Z 258.638,A -85,B 0,C 180,E1 -11314.486,E2 -11314.486} C_VEL
LIN {X 0,Y 397.104,Z 258.641,A -85,B 0,C 180,E1 -11317.084,E2 -11317.084} C_VEL
LIN {X 0,Y 397.142,Z 258.636,A -85,B 0,C 180,E1 -11320.351,E2 -11320.351} C_VEL
LIN {X 0,Y 397.16,Z 258.634,A -85,B 0,C 180,E1 -11323.552,E2 -11323.552} C_VEL
LIN {X 0,Y 397.222,Z 258.628,A -85,B 0,C 180,E1 -11326.701,E2 -11326.701} C_VEL
LIN {X 0,Y 397.211,Z 258.633,A -85,B 0,C 180,E1 -11329.808,E2 -11329.808} C_VEL
LIN {X 0,Y 397.345,Z 258.606,A -85,B 0,C 180,E1 -11332.887,E2 -11332.887} C_VEL
LIN {X 0,Y 397.248,Z 258.627,A -85,B 0,C 180,E1 -11334.924,E2 -11334.924} C_VEL
LIN {X 0,Y 397.443,Z 258.6,A -85,B 0,C 180,E1 -11337.972,E2 -11337.972} C_VEL
LIN {X 0,Y 397.573,Z 258.583,A -85,B 0,C 180,E1 -11339.999,E2 -11339.999} C_VEL
LIN {X 0,Y 397.373,Z 258.611,A -85,B 0,C 180,E1 -11343.04,E2 -11343.04} C_VEL
LIN {X 0,Y 397.336,Z 258.611,A -85,B 0,C 180,E1 -11346.663,E2 -11346.663} C_VEL
LIN {X 0,Y 397.243,Z 258.623,A -85,B 0,C 180,E1 -11349.161,E2 -11349.161} C_VEL
LIN {X 0,Y 397.209,Z 258.63,A -85,B 0,C 180,E1 -11352.257,E2 -11352.257} C_VEL
LIN {X 0,Y 397.168,Z 258.637,A -85,B 0,C 180,E1 -11355.391,E2 -11355.391} C_VEL
LIN {X 0,Y 397.16,Z 258.637,A -85,B 0,C 180,E1 -11358.572,E2 -11358.572} C_VEL
LIN {X 0,Y 397.114,Z 258.641,A -85,B 0,C 180,E1 -11361.816,E2 -11361.816} C_VEL
LIN {X 0,Y 397.14,Z 258.639,A -85,B 0,C 180,E1 -11365.511,E2 -11365.511} C_VEL
LIN {X 0,Y 397.114,Z 258.647,A -85,B 0,C 180,E1 -11368.542,E2 -11368.542} C_VEL
LIN {X 0,Y 397.066,Z 258.643,A -85,B 0,C 180,E1 -11372.071,E2 -11372.071} C_VEL
LIN {X 0,Y 397.106,Z 258.634,A -85,B 0,C 180,E1 -11375.503,E2 -11375.503} C_VEL
LIN {X 0,Y 397.123,Z 258.635,A -85,B 0,C 180,E1 -11378.862,E2 -11378.862} C_VEL
LIN {X 0,Y 397.145,Z 258.635,A -85,B 0,C 180,E1 -11382.255,E2 -11382.255} C_VEL
LIN {X 0,Y 397.137,Z 258.641,A -85,B 0,C 180,E1 -11385.059,E2 -11385.059} C_VEL
LIN {X 0,Y 397.158,Z 258.719,A -85,B 0,C 180,E1 -11387.615,E2 -11387.615} C_VEL
LIN {X 0,Y 399.986,Z 270.784,A -85,B 0,C 180,E1 -11390.763,E2 -11390.763} C_VEL
LIN {X 0,Y 400.172,Z 271.67,A -85,B 0,C 180,E1 -11390.97,E2 -11390.97} C_VEL
LIN {X 0,Y 406.534,Z 286.558,A -85,B 0,C 180,E1 -11391.752,E2 -11391.752} C_VEL
LIN {X 0,Y 409.089,Z 298.164,A -85,B 0,C 180,E1 -11392.167,E2 -11392.167} C_VEL
LIN {X 0,Y 406.992,Z 408.19,A -85,B 0,C 180,E1 -11394.185,E2 -11394.185} C_VEL
LIN {X 0,Y 406.328,Z 422.581,A -85,B 0,C 180,E1 -11394.647,E2 -11394.647} C_VEL
LIN {X 0,Y 405.464,Z 435.816,A -85,B 0,C 180,E1 -11395.263,E2 -11395.263} C_VEL
LIN {X 0,Y 404.516,Z 448.792,A -85,B 0,C 180,E1 -11396.074,E2 -11396.074} C_VEL
LIN {X 0,Y 403.313,Z 461.837,A -85,B 0,C 180,E1 -11397.116,E2 -11397.116} C_VEL
LIN {X 0,Y 402.054,Z 473.059,A -85,B 0,C 180,E1 -11398.225,E2 -11398.225} C_VEL
LIN {X 0,Y 400.827,Z 484.252,A -85,B 0,C 180,E1 -11399.584,E2 -11399.584} C_VEL
LIN {X 0,Y 399.619,Z 494.362,A -85,B 0,C 180,E1 -11401.078,E2 -11401.078} C_VEL
LIN {X 0,Y 398.583,Z 503.436,A -85,B 0,C 180,E1 -11402.714,E2 -11402.714} C_VEL
LIN {X 0,Y 397.756,Z 510.668,A -85,B 0,C 180,E1 -11404.302,E2 -11404.302} C_VEL
LIN {X 0,Y 397.04,Z 516.93,A -85,B 0,C 180,E1 -11405.977,E2 -11405.977} C_VEL
LIN {X 0,Y 396.529,Z 521.922,A -85,B 0,C 180,E1 -11407.631,E2 -11407.631} C_VEL
LIN {X 0,Y 396.16,Z 525.734,A -85,B 0,C 180,E1 -11409.219,E2 -11409.219} C_VEL
LIN {X 0,Y 396.005,Z 527.794,A -85,B 0,C 180,E1 -11410.294,E2 -11410.294} C_VEL
LIN {X 0,Y 395.742,Z 530.741,A -85,B 0,C 180,E1 -11412.429,E2 -11412.429} C_VEL
LIN {X 0,Y 395.641,Z 532.218,A -85,B 0,C 180,E1 -11414.547,E2 -11414.547} C_VEL
LIN {X 0,Y 395.607,Z 532.284,A -85,B 0,C 180,E1 -11416.648,E2 -11416.648} C_VEL
LIN {X 0,Y 395.705,Z 531.787,A -85,B 0,C 180,E1 -11417.695,E2 -11417.695} C_VEL
LIN {X 0,Y 395.697,Z 529.755,A -85,B 0,C 180,E1 -11419.77,E2 -11419.77} C_VEL
LIN {X 0,Y 395.965,Z 526.3,A -85,B 0,C 180,E1 -11421.837,E2 -11421.837} C_VEL
LIN {X 0,Y 396.264,Z 521.36,A -85,B 0,C 180,E1 -11423.892,E2 -11423.892} C_VEL
LIN {X 0,Y 396.709,Z 514.791,A -85,B 0,C 180,E1 -11425.937,E2 -11425.937} C_VEL
LIN {X 0,Y 397.291,Z 507.497,A -85,B 0,C 180,E1 -11427.719,E2 -11427.719} C_VEL
LIN {X 0,Y 397.708,Z 503.341,A -85,B 0,C 180,E1 -11428.579,E2 -11428.579} C_VEL
LIN {X 0,Y 397.399,Z 499.844,A -85,B 0,C 180,E1 -11429.263,E2 -11429.263} C_VEL
LIN {X 0,Y 395.157,Z 493.935,A -85,B 0,C 180,E1 -11430.371,E2 -11430.371} C_VEL
LIN {X 0,Y 392.954,Z 487.594,A -85,B 0,C 180,E1 -11431.434,E2 -11431.434} C_VEL
LIN {X 0,Y 392.702,Z 483.37,A -85,B 0,C 180,E1 -11432.037,E2 -11432.037} C_VEL
LIN {X 0,Y 393.904,Z 471.497,A -85,B 0,C 180,E1 -11433.452,E2 -11433.452} C_VEL
LIN {X 0,Y 394.935,Z 459.864,A -85,B 0,C 180,E1 -11434.58,E2 -11434.58} C_VEL
LIN {X 0,Y 395.944,Z 446.737,A -85,B 0,C 180,E1 -11435.602,E2 -11435.602} C_VEL
LIN {X 0,Y 396.776,Z 433.093,A -85,B 0,C 180,E1 -11436.42,E2 -11436.42} C_VEL
LIN {X 0,Y 397.428,Z 418.701,A -85,B 0,C 180,E1 -11437.047,E2 -11437.047} C_VEL
LIN {X 0,Y 397.919,Z 404.418,A -85,B 0,C 180,E1 -11437.452,E2 -11437.452} C_VEL
LIN {X 0,Y 399.718,Z 298.795,A -85,B 0,C 180,E1 -11439.37,E2 -11439.37} C_VEL
LIN {X 0,Y 395.866,Z 280.45,A -85,B 0,C 180,E1 -11439.929,E2 -11439.929} C_VEL
LIN {X 0,Y 392.568,Z 271.224,A -85,B 0,C 180,E1 -11440.313,E2 -11440.313} C_VEL
LIN {X 0,Y 390.192,Z 259.506,A -85,B 0,C 180,E1 -11443.129,E2 -11443.129} C_VEL
LIN {X 0,Y 390.124,Z 259.511,A -85,B 0,C 180,E1 -11446.752,E2 -11446.752} C_VEL
LIN {X 0,Y 390.106,Z 259.517,A -85,B 0,C 180,E1 -11450.017,E2 -11450.017} C_VEL
LIN {X 0,Y 390.076,Z 259.52,A -85,B 0,C 180,E1 -11453.351,E2 -11453.351} C_VEL
LIN {X 0,Y 390.1,Z 259.514,A -85,B 0,C 180,E1 -11456.769,E2 -11456.769} C_VEL
LIN {X 0,Y 390.039,Z 259.522,A -85,B 0,C 180,E1 -11460.299,E2 -11460.299} C_VEL
LIN {X 0,Y 390.055,Z 259.521,A -85,B 0,C 180,E1 -11464.025,E2 -11464.025} C_VEL
LIN {X 0,Y 390.034,Z 259.528,A -85,B 0,C 180,E1 -11467.552,E2 -11467.552} C_VEL
LIN {X 0,Y 390.07,Z 259.519,A -85,B 0,C 180,E1 -11470.827,E2 -11470.827} C_VEL
LIN {X 0,Y 390.116,Z 259.513,A -85,B 0,C 180,E1 -11473.898,E2 -11473.898} C_VEL
LIN {X 0,Y 390.108,Z 259.516,A -85,B 0,C 180,E1 -11477.614,E2 -11477.614} C_VEL
LIN {X 0,Y 390.083,Z 259.519,A -85,B 0,C 180,E1 -11480.909,E2 -11480.909} C_VEL
LIN {X 0,Y 390.073,Z 259.52,A -85,B 0,C 180,E1 -11484.794,E2 -11484.794} C_VEL
LIN {X 0,Y 390.016,Z 259.525,A -85,B 0,C 180,E1 -11488.497,E2 -11488.497} C_VEL
LIN {X 0,Y 390.106,Z 259.513,A -85,B 0,C 180,E1 -11492.071,E2 -11492.071} C_VEL
LIN {X 0,Y 390.069,Z 259.519,A -85,B 0,C 180,E1 -11495.52,E2 -11495.52} C_VEL
LIN {X 0,Y 390.045,Z 259.528,A -85,B 0,C 180,E1 -11498.879,E2 -11498.879} C_VEL
LIN {X 0,Y 390.118,Z 259.512,A -85,B 0,C 180,E1 -11502.168,E2 -11502.168} C_VEL
LIN {X 0,Y 390.136,Z 259.51,A -85,B 0,C 180,E1 -11505.394,E2 -11505.394} C_VEL
LIN {X 0,Y 390.139,Z 259.514,A -85,B 0,C 180,E1 -11508.572,E2 -11508.572} C_VEL
LIN {X 0,Y 390.299,Z 259.49,A -85,B 0,C 180,E1 -11512.033,E2 -11512.033} C_VEL
LIN {X 0,Y 390.22,Z 259.503,A -85,B 0,C 180,E1 -11514.835,E2 -11514.835} C_VEL
LIN {X 0,Y 390.413,Z 259.476,A -85,B 0,C 180,E1 -11517.938,E2 -11517.938} C_VEL
LIN {X 0,Y 390.542,Z 259.46,A -85,B 0,C 180,E1 -11520.001,E2 -11520.001} C_VEL
LIN {X 0,Y 390.309,Z 259.488,A -85,B 0,C 180,E1 -11523.098,E2 -11523.098} C_VEL
LIN {X 0,Y 390.321,Z 259.491,A -85,B 0,C 180,E1 -11526.203,E2 -11526.203} C_VEL
LIN {X 0,Y 390.199,Z 259.501,A -85,B 0,C 180,E1 -11529.33,E2 -11529.33} C_VEL
LIN {X 0,Y 390.19,Z 259.503,A -85,B 0,C 180,E1 -11533.44,E2 -11533.44} C_VEL
LIN {X 0,Y 390.146,Z 259.508,A -85,B 0,C 180,E1 -11537.31,E2 -11537.31} C_VEL
LIN {X 0,Y 390.083,Z 259.519,A -85,B 0,C 180,E1 -11540.471,E2 -11540.471} C_VEL
LIN {X 0,Y 390.07,Z 259.518,A -85,B 0,C 180,E1 -11543.353,E2 -11543.353} C_VEL
LIN {X 0,Y 390.111,Z 259.513,A -85,B 0,C 180,E1 -11546.77,E2 -11546.77} C_VEL
LIN {X 0,Y 390.042,Z 259.524,A -85,B 0,C 180,E1 -11550.301,E2 -11550.301} C_VEL
LIN {X 0,Y 390.054,Z 259.52,A -85,B 0,C 180,E1 -11552.722,E2 -11552.722} C_VEL
LIN {X 0,Y 390.056,Z 259.526,A -85,B 0,C 180,E1 -11555.827,E2 -11555.827} C_VEL
LIN {X 0,Y 390.071,Z 259.519,A -85,B 0,C 180,E1 -11559.22,E2 -11559.22} C_VEL
LIN {X 0,Y 390.042,Z 259.522,A -85,B 0,C 180,E1 -11562.375,E2 -11562.375} C_VEL
LIN {X 0,Y 390.044,Z 259.524,A -85,B 0,C 180,E1 -11565.355,E2 -11565.355} C_VEL
LIN {X 0,Y 390.031,Z 259.523,A -85,B 0,C 180,E1 -11568.188,E2 -11568.188} C_VEL
LIN {X 0,Y 390.087,Z 259.516,A -85,B 0,C 180,E1 -11570.908,E2 -11570.908} C_VEL
LIN {X 0,Y 390.086,Z 259.516,A -85,B 0,C 180,E1 -11574.794,E2 -11574.794} C_VEL
LIN {X 0,Y 390.03,Z 259.532,A -85,B 0,C 180,E1 -11578.497,E2 -11578.497} C_VEL
LIN {X 0,Y 390.083,Z 259.661,A -85,B 0,C 180,E1 -11579.293,E2 -11579.293} C_VEL
LIN {X 0,Y 392.93,Z 272.304,A -85,B 0,C 180,E1 -11582.047,E2 -11582.047} C_VEL
LIN {X 0,Y 394.566,Z 280.867,A -85,B 0,C 180,E1 -11583.843,E2 -11583.843} C_VEL
LIN {X 0,Y 393.826,Z 291.035,A -85,B 0,C 180,E1 -11585.792,E2 -11585.792} C_VEL
LIN {X 0,Y 399.425,Z 324.203,A -85,B 0,C 180,E1 -11586.731,E2 -11586.731} C_VEL
LIN {X 0,Y 397.72,Z 428.078,A -85,B 0,C 180,E1 -11588.626,E2 -11588.626} C_VEL
LIN {X 0,Y 397.121,Z 442.437,A -85,B 0,C 180,E1 -11589.068,E2 -11589.068} C_VEL
LIN {X 0,Y 396.248,Z 456.246,A -85,B 0,C 180,E1 -11589.698,E2 -11589.698} C_VEL
LIN {X 0,Y 395.332,Z 469.939,A -85,B 0,C 180,E1 -11590.551,E2 -11590.551} C_VEL
LIN {X 0,Y 394.24,Z 482.549,A -85,B 0,C 180,E1 -11591.553,E2 -11591.553} C_VEL
LIN {X 0,Y 393.127,Z 494.268,A -85,B 0,C 180,E1 -11592.71,E2 -11592.71} C_VEL
LIN {X 0,Y 392.134,Z 504.008,A -85,B 0,C 180,E1 -11593.871,E2 -11593.871} C_VEL
LIN {X 0,Y 391.15,Z 514.813,A -85,B 0,C 180,E1 -11595.431,E2 -11595.431} C_VEL
LIN {X 0,Y 390.451,Z 523.725,A -85,B 0,C 180,E1 -11596.998,E2 -11596.998} C_VEL
LIN {X 0,Y 389.66,Z 532.239,A -85,B 0,C 180,E1 -11598.82,E2 -11598.82} C_VEL
LIN {X 0,Y 389.152,Z 539.081,A -85,B 0,C 180,E1 -11600.646,E2 -11600.646} C_VEL
LIN {X 0,Y 388.914,Z 543.772,A -85,B 0,C 180,E1 -11602.211,E2 -11602.211} C_VEL
LIN {X 0,Y 388.753,Z 547.789,A -85,B 0,C 180,E1 -11603.889,E2 -11603.889} C_VEL
LIN {X 0,Y 388.675,Z 551.234,A -85,B 0,C 180,E1 -11605.852,E2 -11605.852} C_VEL
LIN {X 0,Y 388.673,Z 553.498,A -85,B 0,C 180,E1 -11607.927,E2 -11607.927} C_VEL
LIN {X 0,Y 388.708,Z 554.402,A -85,B 0,C 180,E1 -11610,E2 -11610} C_VEL
LIN {X 0,Y 388.657,Z 553.965,A -85,B 0,C 180,E1 -11612.072,E2 -11612.072} C_VEL
LIN {X 0,Y 388.676,Z 552.195,A -85,B 0,C 180,E1 -11614.147,E2 -11614.147} C_VEL
LIN {X 0,Y 388.779,Z 549.055,A -85,B 0,C 180,E1 -11616.226,E2 -11616.226} C_VEL
LIN {X 0,Y 389.036,Z 544.457,A -85,B 0,C 180,E1 -11618.309,E2 -11618.309} C_VEL
LIN {X 0,Y 389.363,Z 539.934,A -85,B 0,C 180,E1 -11619.873,E2 -11619.873} C_VEL
LIN {X 0,Y 390.064,Z 533.44,A -85,B 0,C 180,E1 -11621.694,E2 -11621.694} C_VEL
LIN {X 0,Y 390.721,Z 526.637,A -85,B 0,C 180,E1 -11623.258,E2 -11623.258} C_VEL
LIN {X 0,Y 391.665,Z 518.503,A -85,B 0,C 180,E1 -11624.815,E2 -11624.815} C_VEL
LIN {X 0,Y 392.874,Z 508.729,A -85,B 0,C 180,E1 -11626.364,E2 -11626.364} C_VEL
LIN {X 0,Y 394.274,Z 497.898,A -85,B 0,C 180,E1 -11627.773,E2 -11627.773} C_VEL
LIN {X 0,Y 395.531,Z 487.206,A -85,B 0,C 180,E1 -11628.921,E2 -11628.921} C_VEL
LIN {X 0,Y 396.819,Z 474.642,A -85,B 0,C 180,E1 -11630.026,E2 -11630.026} C_VEL
LIN {X 0,Y 398.051,Z 461.289,A -85,B 0,C 180,E1 -11630.948,E2 -11630.948} C_VEL
LIN {X 0,Y 399.205,Z 447.388,A -85,B 0,C 180,E1 -11631.663,E2 -11631.663} C_VEL
LIN {X 0,Y 399.987,Z 433.842,A -85,B 0,C 180,E1 -11632.161,E2 -11632.161} C_VEL
LIN {X 0,Y 400.518,Z 418.855,A -85,B 0,C 180,E1 -11632.503,E2 -11632.503} C_VEL
LIN {X 0,Y 402.27,Z 324.297,A -85,B 0,C 180,E1 -11634.249,E2 -11634.249} C_VEL
LIN {X 0,Y 398.525,Z 304.735,A -85,B 0,C 180,E1 -11634.922,E2 -11634.922} C_VEL
LIN {X 0,Y 395.415,Z 290.513,A -85,B 0,C 180,E1 -11635.475,E2 -11635.475} C_VEL
LIN {X 0,Y 395.965,Z 285.005,A -85,B 0,C 180,E1 -11636.573,E2 -11636.573} C_VEL
LIN {X 0,Y 393.807,Z 274.305,A -85,B 0,C 180,E1 -11639.016,E2 -11639.016} C_VEL
LIN {X 0,Y 390.995,Z 263.317,A -85,B 0,C 180,E1 -11641.684,E2 -11641.684} C_VEL
LIN {X 0,Y 390.084,Z 259.521,A -85,B 0,C 180,E1 -11642.674,E2 -11642.674} C_VEL
LIN {X 0,Y 390.056,Z 259.53,A -85,B 0,C 180,E1 -11645.824,E2 -11645.824} C_VEL
LIN {X 0,Y 390.069,Z 259.526,A -85,B 0,C 180,E1 -11649.217,E2 -11649.217} C_VEL
LIN {X 0,Y 390.119,Z 259.519,A -85,B 0,C 180,E1 -11652.385,E2 -11652.385} C_VEL
LIN {X 0,Y 390.06,Z 259.521,A -85,B 0,C 180,E1 -11655.355,E2 -11655.355} C_VEL
LIN {X 0,Y 390.029,Z 259.526,A -85,B 0,C 180,E1 -11658.185,E2 -11658.185} C_VEL
LIN {X 0,Y 390.088,Z 259.518,A -85,B 0,C 180,E1 -11660.906,E2 -11660.906} C_VEL
LIN {X 0,Y 390.082,Z 259.502,A -85,B 0,C 180,E1 -11664.792,E2 -11664.792} C_VEL
LIN {X 0,Y 390.023,Z 259.52,A -85,B 0,C 180,E1 -11668.495,E2 -11668.495} C_VEL
LIN {X 0,Y 390.113,Z 259.511,A -85,B 0,C 180,E1 -11672.069,E2 -11672.069} C_VEL
LIN {X 0,Y 390.075,Z 259.518,A -85,B 0,C 180,E1 -11675.518,E2 -11675.518} C_VEL
LIN {X 0,Y 390.05,Z 259.521,A -85,B 0,C 180,E1 -11678.876,E2 -11678.876} C_VEL
LIN {X 0,Y 390.122,Z 259.514,A -85,B 0,C 180,E1 -11682.165,E2 -11682.165} C_VEL
LIN {X 0,Y 390.137,Z 259.511,A -85,B 0,C 180,E1 -11685.391,E2 -11685.391} C_VEL
LIN {X 0,Y 390.142,Z 259.503,A -85,B 0,C 180,E1 -11688.57,E2 -11688.57} C_VEL
LIN {X 0,Y 390.3,Z 259.484,A -85,B 0,C 180,E1 -11692.03,E2 -11692.03} C_VEL
LIN {X 0,Y 390.219,Z 259.502,A -85,B 0,C 180,E1 -11694.832,E2 -11694.832} C_VEL
LIN {X 0,Y 390.412,Z 259.476,A -85,B 0,C 180,E1 -11697.935,E2 -11697.935} C_VEL
LIN {X 0,Y 390.543,Z 259.459,A -85,B 0,C 180,E1 -11699.999,E2 -11699.999} C_VEL
LIN {X 0,Y 390.306,Z 259.492,A -85,B 0,C 180,E1 -11703.095,E2 -11703.095} C_VEL
LIN {X 0,Y 390.291,Z 259.489,A -85,B 0,C 180,E1 -11706.659,E2 -11706.659} C_VEL
LIN {X 0,Y 390.195,Z 259.5,A -85,B 0,C 180,E1 -11709.327,E2 -11709.327} C_VEL
LIN {X 0,Y 390.16,Z 259.51,A -85,B 0,C 180,E1 -11712.482,E2 -11712.482} C_VEL
LIN {X 0,Y 390.128,Z 259.512,A -85,B 0,C 180,E1 -11715.676,E2 -11715.676} C_VEL
LIN {X 0,Y 390.105,Z 259.52,A -85,B 0,C 180,E1 -11718.92,E2 -11718.92} C_VEL
LIN {X 0,Y 390.05,Z 259.523,A -85,B 0,C 180,E1 -11722.232,E2 -11722.232} C_VEL
LIN {X 0,Y 390.106,Z 259.515,A -85,B 0,C 180,E1 -11725.742,E2 -11725.742} C_VEL
LIN {X 0,Y 390.052,Z 259.519,A -85,B 0,C 180,E1 -11729.108,E2 -11729.108} C_VEL
LIN {X 0,Y 390.03,Z 259.527,A -85,B 0,C 180,E1 -11732.721,E2 -11732.721} C_VEL
LIN {X 0,Y 390.044,Z 259.515,A -85,B 0,C 180,E1 -11735.825,E2 -11735.825} C_VEL
LIN {X 0,Y 390.06,Z 259.515,A -85,B 0,C 180,E1 -11739.218,E2 -11739.218} C_VEL
LIN {X 0,Y 390.107,Z 259.512,A -85,B 0,C 180,E1 -11742.386,E2 -11742.386} C_VEL
LIN {X 0,Y 390.105,Z 259.517,A -85,B 0,C 180,E1 -11745.365,E2 -11745.365} C_VEL
LIN {X 0,Y 390.155,Z 259.654,A -85,B 0,C 180,E1 -11747.154,E2 -11747.154} C_VEL
LIN {X 0,Y 393.066,Z 271.951,A -85,B 0,C 180,E1 -11750.406,E2 -11750.406} C_VEL
LIN {X 0,Y 400.478,Z 288.993,A -85,B 0,C 180,E1 -11751.343,E2 -11751.343} C_VEL
LIN {X 0,Y 402.814,Z 299.451,A -85,B 0,C 180,E1 -11751.729,E2 -11751.729} C_VEL
LIN {X 0,Y 400.581,Z 408.193,A -85,B 0,C 180,E1 -11753.75,E2 -11753.75} C_VEL
LIN {X 0,Y 399.926,Z 422.378,A -85,B 0,C 180,E1 -11754.209,E2 -11754.209} C_VEL
LIN {X 0,Y 398.98,Z 435.963,A -85,B 0,C 180,E1 -11754.846,E2 -11754.846} C_VEL
LIN {X 0,Y 397.942,Z 449.352,A -85,B 0,C 180,E1 -11755.699,E2 -11755.699} C_VEL
LIN {X 0,Y 396.753,Z 461.616,A -85,B 0,C 180,E1 -11756.694,E2 -11756.694} C_VEL
LIN {X 0,Y 395.335,Z 473.828,A -85,B 0,C 180,E1 -11757.921,E2 -11757.921} C_VEL
LIN {X 0,Y 394.042,Z 484.921,A -85,B 0,C 180,E1 -11759.301,E2 -11759.301} C_VEL
LIN {X 0,Y 392.77,Z 494.95,A -85,B 0,C 180,E1 -11760.818,E2 -11760.818} C_VEL
LIN {X 0,Y 391.684,Z 503.942,A -85,B 0,C 180,E1 -11762.482,E2 -11762.482} C_VEL
LIN {X 0,Y 390.84,Z 510.865,A -85,B 0,C 180,E1 -11764.034,E2 -11764.034} C_VEL
LIN {X 0,Y 390.145,Z 516.398,A -85,B 0,C 180,E1 -11765.524,E2 -11765.524} C_VEL
LIN {X 0,Y 389.541,Z 521.83,A -85,B 0,C 180,E1 -11767.315,E2 -11767.315} C_VEL
LIN {X 0,Y 389.062,Z 526.608,A -85,B 0,C 180,E1 -11769.376,E2 -11769.376} C_VEL
LIN {X 0,Y 388.788,Z 529.363,A -85,B 0,C 180,E1 -11771.012,E2 -11771.012} C_VEL
LIN {X 0,Y 388.599,Z 531.698,A -85,B 0,C 180,E1 -11773.18,E2 -11773.18} C_VEL
LIN {X 0,Y 388.492,Z 532.596,A -85,B 0,C 180,E1 -11775.33,E2 -11775.33} C_VEL
LIN {X 0,Y 388.603,Z 532.046,A -85,B 0,C 180,E1 -11777.572,E2 -11777.572} C_VEL
LIN {X 0,Y 388.613,Z 530.226,A -85,B 0,C 180,E1 -11779.581,E2 -11779.581} C_VEL
LIN {X 0,Y 388.851,Z 526.924,A -85,B 0,C 180,E1 -11781.687,E2 -11781.687} C_VEL
LIN {X 0,Y 389.153,Z 522.123,A -85,B 0,C 180,E1 -11783.78,E2 -11783.78} C_VEL
LIN {X 0,Y 389.613,Z 515.698,A -85,B 0,C 180,E1 -11785.863,E2 -11785.863} C_VEL
LIN {X 0,Y 390.174,Z 508.566,A -85,B 0,C 180,E1 -11787.677,E2 -11787.677} C_VEL
LIN {X 0,Y 390.929,Z 501.095,A -85,B 0,C 180,E1 -11789.228,E2 -11789.228} C_VEL
LIN {X 0,Y 391.862,Z 492.136,A -85,B 0,C 180,E1 -11790.771,E2 -11790.771} C_VEL
LIN {X 0,Y 392.702,Z 483.37,A -85,B 0,C 180,E1 -11792.037,E2 -11792.037} C_VEL
LIN {X 0,Y 392.472,Z 479.03,A -85,B 0,C 180,E1 -11792.619,E2 -11792.619} C_VEL
LIN {X 0,Y 390.395,Z 471.788,A -85,B 0,C 180,E1 -11793.571,E2 -11793.571} C_VEL
LIN {X 0,Y 388.354,Z 464.194,A -85,B 0,C 180,E1 -11794.459,E2 -11794.459} C_VEL
LIN {X 0,Y 388.169,Z 459.246,A -85,B 0,C 180,E1 -11794.933,E2 -11794.933} C_VEL
LIN {X 0,Y 389.223,Z 446.045,A -85,B 0,C 180,E1 -11795.959,E2 -11795.959} C_VEL
LIN {X 0,Y 390.008,Z 433.361,A -85,B 0,C 180,E1 -11796.727,E2 -11796.727} C_VEL
LIN {X 0,Y 390.703,Z 418.984,A -85,B 0,C 180,E1 -11797.364,E2 -11797.364} C_VEL
LIN {X 0,Y 391.197,Z 404.777,A -85,B 0,C 180,E1 -11797.776,E2 -11797.776} C_VEL
LIN {X 0,Y 392.97,Z 299.022,A -85,B 0,C 180,E1 -11799.731,E2 -11799.731} C_VEL
LIN {X 0,Y 389.193,Z 281.846,A -85,B 0,C 180,E1 -11800.276,E2 -11800.276} C_VEL
LIN {X 0,Y 385.378,Z 271.378,A -85,B 0,C 180,E1 -11800.73,E2 -11800.73} C_VEL
LIN {X 0,Y 383.137,Z 260.385,A -85,B 0,C 180,E1 -11803.461,E2 -11803.461} C_VEL
LIN {X 0,Y 383.082,Z 260.391,A -85,B 0,C 180,E1 -11807.455,E2 -11807.455} C_VEL
LIN {X 0,Y 383.03,Z 260.394,A -85,B 0,C 180,E1 -11810.653,E2 -11810.653} C_VEL
LIN {X 0,Y 383.02,Z 260.401,A -85,B 0,C 180,E1 -11813.808,E2 -11813.808} C_VEL
LIN {X 0,Y 383.067,Z 260.392,A -85,B 0,C 180,E1 -11816.124,E2 -11816.124} C_VEL
LIN {X 0,Y 383.038,Z 260.393,A -85,B 0,C 180,E1 -11818.492,E2 -11818.492} C_VEL
LIN {X 0,Y 383,Z 260.399,A -85,B 0,C 180,E1 -11822.15,E2 -11822.15} C_VEL
LIN {X 0,Y 383.005,Z 260.398,A -85,B 0,C 180,E1 -11824.669,E2 -11824.669} C_VEL
LIN {X 0,Y 382.99,Z 260.401,A -85,B 0,C 180,E1 -11827.905,E2 -11827.905} C_VEL
LIN {X 0,Y 383.034,Z 260.4,A -85,B 0,C 180,E1 -11831.34,E2 -11831.34} C_VEL
LIN {X 0,Y 383.058,Z 260.391,A -85,B 0,C 180,E1 -11834.316,E2 -11834.316} C_VEL
LIN {X 0,Y 383.063,Z 260.397,A -85,B 0,C 180,E1 -11837.25,E2 -11837.25} C_VEL
LIN {X 0,Y 383.01,Z 260.397,A -85,B 0,C 180,E1 -11840.413,E2 -11840.413} C_VEL
LIN {X 0,Y 383.014,Z 260.396,A -85,B 0,C 180,E1 -11844.046,E2 -11844.046} C_VEL
LIN {X 0,Y 382.976,Z 260.403,A -85,B 0,C 180,E1 -11847.579,E2 -11847.579} C_VEL
LIN {X 0,Y 382.986,Z 260.4,A -85,B 0,C 180,E1 -11850.302,E2 -11850.302} C_VEL
LIN {X 0,Y 383.046,Z 260.396,A -85,B 0,C 180,E1 -11852.699,E2 -11852.699} C_VEL
LIN {X 0,Y 383.041,Z 260.399,A -85,B 0,C 180,E1 -11855.041,E2 -11855.041} C_VEL
LIN {X 0,Y 382.982,Z 260.403,A -85,B 0,C 180,E1 -11858.47,E2 -11858.47} C_VEL
LIN {X 0,Y 383.053,Z 260.391,A -85,B 0,C 180,E1 -11861.828,E2 -11861.828} C_VEL
LIN {X 0,Y 383.102,Z 260.388,A -85,B 0,C 180,E1 -11865.12,E2 -11865.12} C_VEL
LIN {X 0,Y 383.088,Z 260.39,A -85,B 0,C 180,E1 -11868.359,E2 -11868.359} C_VEL
LIN {X 0,Y 383.256,Z 260.367,A -85,B 0,C 180,E1 -11871.977,E2 -11871.977} C_VEL
LIN {X 0,Y 383.192,Z 260.379,A -85,B 0,C 180,E1 -11874.74,E2 -11874.74} C_VEL
LIN {X 0,Y 383.38,Z 260.352,A -85,B 0,C 180,E1 -11877.9,E2 -11877.9} C_VEL
LIN {X 0,Y 383.512,Z 260.336,A -85,B 0,C 180,E1 -11880.001,E2 -11880.001} C_VEL
LIN {X 0,Y 383.245,Z 260.368,A -85,B 0,C 180,E1 -11883.155,E2 -11883.155} C_VEL
LIN {X 0,Y 383.277,Z 260.37,A -85,B 0,C 180,E1 -11886.318,E2 -11886.318} C_VEL
LIN {X 0,Y 383.146,Z 260.38,A -85,B 0,C 180,E1 -11889.504,E2 -11889.504} C_VEL
LIN {X 0,Y 383.121,Z 260.384,A -85,B 0,C 180,E1 -11893.537,E2 -11893.537} C_VEL
LIN {X 0,Y 383.092,Z 260.387,A -85,B 0,C 180,E1 -11897.456,E2 -11897.456} C_VEL
LIN {X 0,Y 383.025,Z 260.397,A -85,B 0,C 180,E1 -11900.648,E2 -11900.648} C_VEL
LIN {X 0,Y 383.022,Z 260.399,A -85,B 0,C 180,E1 -11903.809,E2 -11903.809} C_VEL
LIN {X 0,Y 383.077,Z 260.394,A -85,B 0,C 180,E1 -11906.125,E2 -11906.125} C_VEL
LIN {X 0,Y 383.047,Z 260.394,A -85,B 0,C 180,E1 -11908.493,E2 -11908.493} C_VEL
LIN {X 0,Y 383.006,Z 260.399,A -85,B 0,C 180,E1 -11912.428,E2 -11912.428} C_VEL
LIN {X 0,Y 383.025,Z 260.4,A -85,B 0,C 180,E1 -11915.957,E2 -11915.957} C_VEL
LIN {X 0,Y 383.016,Z 260.401,A -85,B 0,C 180,E1 -11919.588,E2 -11919.588} C_VEL
LIN {X 0,Y 383.005,Z 260.397,A -85,B 0,C 180,E1 -11922.78,E2 -11922.78} C_VEL
LIN {X 0,Y 382.997,Z 260.404,A -85,B 0,C 180,E1 -11925.79,E2 -11925.79} C_VEL
LIN {X 0,Y 382.988,Z 260.4,A -85,B 0,C 180,E1 -11928.797,E2 -11928.797} C_VEL
LIN {X 0,Y 382.998,Z 260.4,A -85,B 0,C 180,E1 -11932.098,E2 -11932.098} C_VEL
LIN {X 0,Y 383.02,Z 260.401,A -85,B 0,C 180,E1 -11935.333,E2 -11935.333} C_VEL
LIN {X 0,Y 383.037,Z 260.517,A -85,B 0,C 180,E1 -11938.972,E2 -11938.972} C_VEL
LIN {X 0,Y 386.149,Z 274.411,A -85,B 0,C 180,E1 -11942.054,E2 -11942.054} C_VEL
LIN {X 0,Y 387.587,Z 281.758,A -85,B 0,C 180,E1 -11943.625,E2 -11943.625} C_VEL
LIN {X 0,Y 387.013,Z 291.125,A -85,B 0,C 180,E1 -11945.415,E2 -11945.415} C_VEL
LIN {X 0,Y 392.763,Z 325.29,A -85,B 0,C 180,E1 -11946.399,E2 -11946.399} C_VEL
LIN {X 0,Y 390.982,Z 428.283,A -85,B 0,C 180,E1 -11948.308,E2 -11948.308} C_VEL
LIN {X 0,Y 390.369,Z 442.455,A -85,B 0,C 180,E1 -11948.758,E2 -11948.758} C_VEL
LIN {X 0,Y 389.457,Z 456.205,A -85,B 0,C 180,E1 -11949.397,E2 -11949.397} C_VEL
LIN {X 0,Y 388.608,Z 468.976,A -85,B 0,C 180,E1 -11950.2,E2 -11950.2} C_VEL
LIN {X 0,Y 387.437,Z 481.728,A -85,B 0,C 180,E1 -11951.218,E2 -11951.218} C_VEL
LIN {X 0,Y 386.284,Z 493.557,A -85,B 0,C 180,E1 -11952.394,E2 -11952.394} C_VEL
LIN {X 0,Y 385.256,Z 503.385,A -85,B 0,C 180,E1 -11953.575,E2 -11953.575} C_VEL
LIN {X 0,Y 384.185,Z 514.257,A -85,B 0,C 180,E1 -11955.161,E2 -11955.161} C_VEL
LIN {X 0,Y 383.475,Z 523.231,A -85,B 0,C 180,E1 -11956.757,E2 -11956.757} C_VEL
LIN {X 0,Y 382.648,Z 531.8,A -85,B 0,C 180,E1 -11958.613,E2 -11958.613} C_VEL
LIN {X 0,Y 382.096,Z 538.693,A -85,B 0,C 180,E1 -11960.472,E2 -11960.472} C_VEL
LIN {X 0,Y 381.841,Z 543.426,A -85,B 0,C 180,E1 -11962.066,E2 -11962.066} C_VEL
LIN {X 0,Y 381.66,Z 547.784,A -85,B 0,C 180,E1 -11963.924,E2 -11963.924} C_VEL
LIN {X 0,Y 381.6,Z 550.963,A -85,B 0,C 180,E1 -11965.775,E2 -11965.775} C_VEL
LIN {X 0,Y 381.572,Z 553.258,A -85,B 0,C 180,E1 -11967.889,E2 -11967.889} C_VEL
LIN {X 0,Y 381.639,Z 554.194,A -85,B 0,C 180,E1 -11970,E2 -11970} C_VEL
LIN {X 0,Y 381.555,Z 553.788,A -85,B 0,C 180,E1 -11972.111,E2 -11972.111} C_VEL
LIN {X 0,Y 381.601,Z 552.051,A -85,B 0,C 180,E1 -11974.225,E2 -11974.225} C_VEL
LIN {X 0,Y 381.705,Z 548.947,A -85,B 0,C 180,E1 -11976.342,E2 -11976.342} C_VEL
LIN {X 0,Y 381.975,Z 544.395,A -85,B 0,C 180,E1 -11978.464,E2 -11978.464} C_VEL
LIN {X 0,Y 382.326,Z 539.901,A -85,B 0,C 180,E1 -11980.057,E2 -11980.057} C_VEL
LIN {X 0,Y 383.093,Z 533.448,A -85,B 0,C 180,E1 -11981.91,E2 -11981.91} C_VEL
LIN {X 0,Y 383.924,Z 525.461,A -85,B 0,C 180,E1 -11983.767,E2 -11983.767} C_VEL
LIN {X 0,Y 384.972,Z 517.128,A -85,B 0,C 180,E1 -11985.349,E2 -11985.349} C_VEL
LIN {X 0,Y 386.283,Z 507.13,A -85,B 0,C 180,E1 -11986.923,E2 -11986.923} C_VEL
LIN {X 0,Y 387.814,Z 496.019,A -85,B 0,C 180,E1 -11988.352,E2 -11988.352} C_VEL
LIN {X 0,Y 389.137,Z 485.004,A -85,B 0,C 180,E1 -11989.518,E2 -11989.518} C_VEL
LIN {X 0,Y 390.408,Z 473.157,A -85,B 0,C 180,E1 -11990.543,E2 -11990.543} C_VEL
LIN {X 0,Y 391.659,Z 459.929,A -85,B 0,C 180,E1 -11991.445,E2 -11991.445} C_VEL
LIN {X 0,Y 392.836,Z 446.327,A -85,B 0,C 180,E1 -11992.136,E2 -11992.136} C_VEL
LIN {X 0,Y 393.68,Z 432.352,A -85,B 0,C 180,E1 -11992.639,E2 -11992.639} C_VEL
LIN {X 0,Y 394.268,Z 413.174,A -85,B 0,C 180,E1 -11993.054,E2 -11993.054} C_VEL
LIN {X 0,Y 396.042,Z 326.138,A -85,B 0,C 180,E1 -11994.68,E2 -11994.68} C_VEL
LIN {X 0,Y 392.951,Z 309.115,A -85,B 0,C 180,E1 -11995.268,E2 -11995.268} C_VEL
LIN {X 0,Y 388.839,Z 290.242,A -85,B 0,C 180,E1 -11996.026,E2 -11996.026} C_VEL
LIN {X 0,Y 389.114,Z 286.297,A -85,B 0,C 180,E1 -11996.842,E2 -11996.842} C_VEL
LIN {X 0,Y 386.898,Z 275.708,A -85,B 0,C 180,E1 -11999.316,E2 -11999.316} C_VEL
LIN {X 0,Y 383.893,Z 263.761,A -85,B 0,C 180,E1 -12002.295,E2 -12002.295} C_VEL
LIN {X 0,Y 383.016,Z 260.406,A -85,B 0,C 180,E1 -12003.206,E2 -12003.206} C_VEL
LIN {X 0,Y 383.032,Z 260.408,A -85,B 0,C 180,E1 -12006.163,E2 -12006.163} C_VEL
LIN {X 0,Y 383.015,Z 260.399,A -85,B 0,C 180,E1 -12009.956,E2 -12009.956} C_VEL
LIN {X 0,Y 383.065,Z 260.395,A -85,B 0,C 180,E1 -12012.787,E2 -12012.787} C_VEL
LIN {X 0,Y 383.006,Z 260.4,A -85,B 0,C 180,E1 -12015.789,E2 -12015.789} C_VEL
LIN {X 0,Y 382.986,Z 260.404,A -85,B 0,C 180,E1 -12018.795,E2 -12018.795} C_VEL
LIN {X 0,Y 382.997,Z 260.401,A -85,B 0,C 180,E1 -12022.095,E2 -12022.095} C_VEL
LIN {X 0,Y 383.015,Z 260.386,A -85,B 0,C 180,E1 -12025.331,E2 -12025.331} C_VEL
LIN {X 0,Y 382.983,Z 260.396,A -85,B 0,C 180,E1 -12029.08,E2 -12029.08} C_VEL
LIN {X 0,Y 383.053,Z 260.39,A -85,B 0,C 180,E1 -12032.697,E2 -12032.697} C_VEL
LIN {X 0,Y 383.029,Z 260.393,A -85,B 0,C 180,E1 -12036.191,E2 -12036.191} C_VEL
LIN {X 0,Y 383.05,Z 260.391,A -85,B 0,C 180,E1 -12039.597,E2 -12039.597} C_VEL
LIN {X 0,Y 383.099,Z 260.387,A -85,B 0,C 180,E1 -12042.93,E2 -12042.93} C_VEL
LIN {X 0,Y 383.119,Z 260.385,A -85,B 0,C 180,E1 -12046.462,E2 -12046.462} C_VEL
LIN {X 0,Y 383.145,Z 260.382,A -85,B 0,C 180,E1 -12050.496,E2 -12050.496} C_VEL
LIN {X 0,Y 383.275,Z 260.366,A -85,B 0,C 180,E1 -12053.682,E2 -12053.682} C_VEL
LIN {X 0,Y 383.379,Z 260.353,A -85,B 0,C 180,E1 -12057.897,E2 -12057.897} C_VEL
LIN {X 0,Y 383.512,Z 260.334,A -85,B 0,C 180,E1 -12059.999,E2 -12059.999} C_VEL
LIN {X 0,Y 383.243,Z 260.373,A -85,B 0,C 180,E1 -12063.152,E2 -12063.152} C_VEL
LIN {X 0,Y 383.25,Z 260.365,A -85,B 0,C 180,E1 -12066.651,E2 -12066.651} C_VEL
LIN {X 0,Y 383.141,Z 260.377,A -85,B 0,C 180,E1 -12069.501,E2 -12069.501} C_VEL
LIN {X 0,Y 383.115,Z 260.381,A -85,B 0,C 180,E1 -12073.535,E2 -12073.535} C_VEL
LIN {X 0,Y 383.084,Z 260.387,A -85,B 0,C 180,E1 -12077.454,E2 -12077.454} C_VEL
LIN {X 0,Y 383.036,Z 260.394,A -85,B 0,C 180,E1 -12080.653,E2 -12080.653} C_VEL
LIN {X 0,Y 383.03,Z 260.392,A -85,B 0,C 180,E1 -12083.806,E2 -12083.806} C_VEL
LIN {X 0,Y 383.044,Z 260.396,A -85,B 0,C 180,E1 -12087.301,E2 -12087.301} C_VEL
LIN {X 0,Y 382.973,Z 260.391,A -85,B 0,C 180,E1 -12090.917,E2 -12090.917} C_VEL
LIN {X 0,Y 383.005,Z 260.391,A -85,B 0,C 180,E1 -12094.667,E2 -12094.667} C_VEL
LIN {X 0,Y 382.99,Z 260.403,A -85,B 0,C 180,E1 -12097.904,E2 -12097.904} C_VEL
LIN {X 0,Y 383.033,Z 260.397,A -85,B 0,C 180,E1 -12101.338,E2 -12101.338} C_VEL
LIN {X 0,Y 383.056,Z 260.396,A -85,B 0,C 180,E1 -12104.314,E2 -12104.314} C_VEL
LIN {X 0,Y 383.107,Z 260.517,A -85,B 0,C 180,E1 -12106.636,E2 -12106.636} C_VEL
LIN {X 0,Y 385.912,Z 272.082,A -85,B 0,C 180,E1 -12109.807,E2 -12109.807} C_VEL
LIN {X 0,Y 394.489,Z 291.468,A -85,B 0,C 180,E1 -12110.924,E2 -12110.924} C_VEL
LIN {X 0,Y 396.447,Z 300.224,A -85,B 0,C 180,E1 -12111.258,E2 -12111.258} C_VEL
LIN {X 0,Y 394.755,Z 382.904,A -85,B 0,C 180,E1 -12112.805,E2 -12112.805} C_VEL
LIN {X 0,Y 394.117,Z 409.848,A -85,B 0,C 180,E1 -12113.345,E2 -12113.345} C_VEL
LIN {X 0,Y 393.402,Z 424.233,A -85,B 0,C 180,E1 -12113.84,E2 -12113.84} C_VEL
LIN {X 0,Y 392.464,Z 437.392,A -85,B 0,C 180,E1 -12114.489,E2 -12114.489} C_VEL
LIN {X 0,Y 391.362,Z 450.47,A -85,B 0,C 180,E1 -12115.35,E2 -12115.35} C_VEL
LIN {X 0,Y 390.104,Z 462.574,A -85,B 0,C 180,E1 -12116.36,E2 -12116.36} C_VEL
LIN {X 0,Y 388.621,Z 474.637,A -85,B 0,C 180,E1 -12117.606,E2 -12117.606} C_VEL
LIN {X 0,Y 387.411,Z 484.61,A -85,B 0,C 180,E1 -12118.872,E2 -12118.872} C_VEL
LIN {X 0,Y 386.145,Z 493.831,A -85,B 0,C 180,E1 -12120.268,E2 -12120.268} C_VEL
LIN {X 0,Y 384.937,Z 503.057,A -85,B 0,C 180,E1 -12121.958,E2 -12121.958} C_VEL
LIN {X 0,Y 383.898,Z 511.114,A -85,B 0,C 180,E1 -12123.767,E2 -12123.767} C_VEL
LIN {X 0,Y 383.056,Z 517.76,A -85,B 0,C 180,E1 -12125.619,E2 -12125.619} C_VEL
LIN {X 0,Y 382.485,Z 522.578,A -85,B 0,C 180,E1 -12127.303,E2 -12127.303} C_VEL
LIN {X 0,Y 382.071,Z 526.384,A -85,B 0,C 180,E1 -12128.981,E2 -12128.981} C_VEL
LIN {X 0,Y 381.771,Z 529.277,A -85,B 0,C 180,E1 -12130.649,E2 -12130.649} C_VEL
LIN {X 0,Y 381.519,Z 531.742,A -85,B 0,C 180,E1 -12132.859,E2 -12132.859} C_VEL
LIN {X 0,Y 381.397,Z 532.767,A -85,B 0,C 180,E1 -12135.05,E2 -12135.05} C_VEL
LIN {X 0,Y 381.482,Z 532.393,A -85,B 0,C 180,E1 -12137.228,E2 -12137.228} C_VEL
LIN {X 0,Y 381.506,Z 530.646,A -85,B 0,C 180,E1 -12139.385,E2 -12139.385} C_VEL
LIN {X 0,Y 381.724,Z 527.502,A -85,B 0,C 180,E1 -12141.53,E2 -12141.53} C_VEL
LIN {X 0,Y 382.01,Z 523.458,A -85,B 0,C 180,E1 -12143.424,E2 -12143.424} C_VEL
LIN {X 0,Y 382.337,Z 518.329,A -85,B 0,C 180,E1 -12145.255,E2 -12145.255} C_VEL
LIN {X 0,Y 382.882,Z 511.784,A -85,B 0,C 180,E1 -12147.107,E2 -12147.107} C_VEL
LIN {X 0,Y 383.714,Z 503.666,A -85,B 0,C 180,E1 -12148.951,E2 -12148.951} C_VEL
LIN {X 0,Y 384.604,Z 495.184,A -85,B 0,C 180,E1 -12150.524,E2 -12150.524} C_VEL
LIN {X 0,Y 385.645,Z 484.938,A -85,B 0,C 180,E1 -12152.089,E2 -12152.089} C_VEL
LIN {X 0,Y 386.87,Z 473.471,A -85,B 0,C 180,E1 -12153.515,E2 -12153.515} C_VEL
LIN {X 0,Y 388.036,Z 460.744,A -85,B 0,C 180,E1 -12154.798,E2 -12154.798} C_VEL
LIN {X 0,Y 388.169,Z 459.246,A -85,B 0,C 180,E1 -12154.933,E2 -12154.933} C_VEL
LIN {X 0,Y 387.976,Z 454.174,A -85,B 0,C 180,E1 -12155.386,E2 -12155.386} C_VEL
LIN {X 0,Y 385.724,Z 445.894,A -85,B 0,C 180,E1 -12156.135,E2 -12156.135} C_VEL
LIN {X 0,Y 383.542,Z 437.347,A -85,B 0,C 180,E1 -12156.807,E2 -12156.807} C_VEL
LIN {X 0,Y 383.339,Z 431.867,A -85,B 0,C 180,E1 -12157.129,E2 -12157.129} C_VEL
LIN {X 0,Y 384.066,Z 417.314,A -85,B 0,C 180,E1 -12157.756,E2 -12157.756} C_VEL
LIN {X 0,Y 384.48,Z 403.462,A -85,B 0,C 180,E1 -12158.144,E2 -12158.144} C_VEL
LIN {X 0,Y 386.338,Z 300.029,A -85,B 0,C 180,E1 -12160.081,E2 -12160.081} C_VEL
LIN {X 0,Y 382.888,Z 284.345,A -85,B 0,C 180,E1 -12160.59,E2 -12160.59} C_VEL
LIN {X 0,Y 378.21,Z 271.624,A -85,B 0,C 180,E1 -12161.145,E2 -12161.145} C_VEL
LIN {X 0,Y 376.092,Z 261.264,A -85,B 0,C 180,E1 -12163.735,E2 -12163.735} C_VEL
LIN {X 0,Y 376.031,Z 261.271,A -85,B 0,C 180,E1 -12167.608,E2 -12167.608} C_VEL
LIN {X 0,Y 375.993,Z 261.271,A -85,B 0,C 180,E1 -12170.844,E2 -12170.844} C_VEL
LIN {X 0,Y 375.98,Z 261.274,A -85,B 0,C 180,E1 -12174.282,E2 -12174.282} C_VEL
LIN {X 0,Y 376.006,Z 261.269,A -85,B 0,C 180,E1 -12176.653,E2 -12176.653} C_VEL
LIN {X 0,Y 375.968,Z 261.276,A -85,B 0,C 180,E1 -12179.079,E2 -12179.079} C_VEL
LIN {X 0,Y 375.937,Z 261.279,A -85,B 0,C 180,E1 -12182.829,E2 -12182.829} C_VEL
LIN {X 0,Y 375.945,Z 261.283,A -85,B 0,C 180,E1 -12185.416,E2 -12185.416} C_VEL
LIN {X 0,Y 375.965,Z 261.275,A -85,B 0,C 180,E1 -12188.272,E2 -12188.272} C_VEL
LIN {X 0,Y 375.977,Z 261.277,A -85,B 0,C 180,E1 -12191.611,E2 -12191.611} C_VEL
LIN {X 0,Y 376.002,Z 261.276,A -85,B 0,C 180,E1 -12195.256,E2 -12195.256} C_VEL
LIN {X 0,Y 375.988,Z 261.277,A -85,B 0,C 180,E1 -12199.142,E2 -12199.142} C_VEL
LIN {X 0,Y 375.956,Z 261.276,A -85,B 0,C 180,E1 -12201.913,E2 -12201.913} C_VEL
LIN {X 0,Y 375.968,Z 261.278,A -85,B 0,C 180,E1 -12205.334,E2 -12205.334} C_VEL
LIN {X 0,Y 375.948,Z 261.277,A -85,B 0,C 180,E1 -12208.439,E2 -12208.439} C_VEL
LIN {X 0,Y 375.991,Z 261.271,A -85,B 0,C 180,E1 -12212.143,E2 -12212.143} C_VEL
LIN {X 0,Y 375.995,Z 261.273,A -85,B 0,C 180,E1 -12214.54,E2 -12214.54} C_VEL
LIN {X 0,Y 375.952,Z 261.276,A -85,B 0,C 180,E1 -12218.047,E2 -12218.047} C_VEL
LIN {X 0,Y 375.999,Z 261.271,A -85,B 0,C 180,E1 -12221.474,E2 -12221.474} C_VEL
LIN {X 0,Y 376.05,Z 261.27,A -85,B 0,C 180,E1 -12224.834,E2 -12224.834} C_VEL
LIN {X 0,Y 376.041,Z 261.266,A -85,B 0,C 180,E1 -12228.138,E2 -12228.138} C_VEL
LIN {X 0,Y 376.211,Z 261.244,A -85,B 0,C 180,E1 -12231.92,E2 -12231.92} C_VEL
LIN {X 0,Y 376.164,Z 261.256,A -85,B 0,C 180,E1 -12234.641,E2 -12234.641} C_VEL
LIN {X 0,Y 376.347,Z 261.228,A -85,B 0,C 180,E1 -12237.861,E2 -12237.861} C_VEL
LIN {X 0,Y 376.481,Z 261.212,A -85,B 0,C 180,E1 -12240.001,E2 -12240.001} C_VEL
LIN {X 0,Y 376.183,Z 261.248,A -85,B 0,C 180,E1 -12243.214,E2 -12243.214} C_VEL
LIN {X 0,Y 376.235,Z 261.247,A -85,B 0,C 180,E1 -12246.437,E2 -12246.437} C_VEL
LIN {X 0,Y 376.113,Z 261.257,A -85,B 0,C 180,E1 -12249.683,E2 -12249.683} C_VEL
LIN {X 0,Y 376.085,Z 261.261,A -85,B 0,C 180,E1 -12253.659,E2 -12253.659} C_VEL
LIN {X 0,Y 376.041,Z 261.266,A -85,B 0,C 180,E1 -12257.609,E2 -12257.609} C_VEL
LIN {X 0,Y 375.975,Z 261.274,A -85,B 0,C 180,E1 -12260.834,E2 -12260.834} C_VEL
LIN {X 0,Y 375.986,Z 261.276,A -85,B 0,C 180,E1 -12264.283,E2 -12264.283} C_VEL
LIN {X 0,Y 376.017,Z 261.269,A -85,B 0,C 180,E1 -12266.654,E2 -12266.654} C_VEL
LIN {X 0,Y 375.974,Z 261.273,A -85,B 0,C 180,E1 -12269.08,E2 -12269.08} C_VEL
LIN {X 0,Y 375.955,Z 261.276,A -85,B 0,C 180,E1 -12272.829,E2 -12272.829} C_VEL
LIN {X 0,Y 375.957,Z 261.278,A -85,B 0,C 180,E1 -12275.417,E2 -12275.417} C_VEL
LIN {X 0,Y 375.975,Z 261.275,A -85,B 0,C 180,E1 -12278.272,E2 -12278.272} C_VEL
LIN {X 0,Y 375.934,Z 261.284,A -85,B 0,C 180,E1 -12281.602,E2 -12281.602} C_VEL
LIN {X 0,Y 375.927,Z 261.282,A -85,B 0,C 180,E1 -12285.27,E2 -12285.27} C_VEL
LIN {X 0,Y 375.935,Z 261.279,A -85,B 0,C 180,E1 -12288.401,E2 -12288.401} C_VEL
LIN {X 0,Y 375.973,Z 261.278,A -85,B 0,C 180,E1 -12291.731,E2 -12291.731} C_VEL
LIN {X 0,Y 375.982,Z 261.277,A -85,B 0,C 180,E1 -12295.334,E2 -12295.334} C_VEL
LIN {X 0,Y 376.005,Z 261.485,A -85,B 0,C 180,E1 -12298.663,E2 -12298.663} C_VEL
LIN {X 0,Y 379.087,Z 275.271,A -85,B 0,C 180,E1 -12301.788,E2 -12301.788} C_VEL
LIN {X 0,Y 380.592,Z 282.705,A -85,B 0,C 180,E1 -12303.411,E2 -12303.411} C_VEL
LIN {X 0,Y 380.362,Z 288.401,A -85,B 0,C 180,E1 -12304.559,E2 -12304.559} C_VEL
LIN {X 0,Y 380.164,Z 290.551,A -85,B 0,C 180,E1 -12304.984,E2 -12304.984} C_VEL
LIN {X 0,Y 386.094,Z 326.154,A -85,B 0,C 180,E1 -12306.052,E2 -12306.052} C_VEL
LIN {X 0,Y 384.247,Z 428.304,A -85,B 0,C 180,E1 -12307.979,E2 -12307.979} C_VEL
LIN {X 0,Y 383.629,Z 442.395,A -85,B 0,C 180,E1 -12308.436,E2 -12308.436} C_VEL
LIN {X 0,Y 382.679,Z 456.115,A -85,B 0,C 180,E1 -12309.086,E2 -12309.086} C_VEL
LIN {X 0,Y 381.739,Z 469.389,A -85,B 0,C 180,E1 -12309.94,E2 -12309.94} C_VEL
LIN {X 0,Y 380.529,Z 482.338,A -85,B 0,C 180,E1 -12311.003,E2 -12311.003} C_VEL
LIN {X 0,Y 379.331,Z 494.032,A -85,B 0,C 180,E1 -12312.2,E2 -12312.2} C_VEL
LIN {X 0,Y 378.162,Z 504.735,A -85,B 0,C 180,E1 -12313.536,E2 -12313.536} C_VEL
LIN {X 0,Y 377.101,Z 515.353,A -85,B 0,C 180,E1 -12315.152,E2 -12315.152} C_VEL
LIN {X 0,Y 376.352,Z 524.254,A -85,B 0,C 180,E1 -12316.805,E2 -12316.805} C_VEL
LIN {X 0,Y 375.529,Z 532.468,A -85,B 0,C 180,E1 -12318.667,E2 -12318.667} C_VEL
LIN {X 0,Y 375.049,Z 538.297,A -85,B 0,C 180,E1 -12320.291,E2 -12320.291} C_VEL
LIN {X 0,Y 374.766,Z 543.073,A -85,B 0,C 180,E1 -12321.915,E2 -12321.915} C_VEL
LIN {X 0,Y 374.571,Z 547.763,A -85,B 0,C 180,E1 -12323.955,E2 -12323.955} C_VEL
LIN {X 0,Y 374.504,Z 550.686,A -85,B 0,C 180,E1 -12325.695,E2 -12325.695} C_VEL
LIN {X 0,Y 374.471,Z 553.016,A -85,B 0,C 180,E1 -12327.849,E2 -12327.849} C_VEL
LIN {X 0,Y 374.554,Z 553.986,A -85,B 0,C 180,E1 -12330,E2 -12330} C_VEL
LIN {X 0,Y 374.453,Z 553.613,A -85,B 0,C 180,E1 -12332.151,E2 -12332.151} C_VEL
LIN {X 0,Y 374.506,Z 551.909,A -85,B 0,C 180,E1 -12334.305,E2 -12334.305} C_VEL
LIN {X 0,Y 374.625,Z 548.84,A -85,B 0,C 180,E1 -12336.463,E2 -12336.463} C_VEL
LIN {X 0,Y 374.93,Z 544.326,A -85,B 0,C 180,E1 -12338.624,E2 -12338.624} C_VEL
LIN {X 0,Y 375.3,Z 539.868,A -85,B 0,C 180,E1 -12340.247,E2 -12340.247} C_VEL
LIN {X 0,Y 376.12,Z 533.463,A -85,B 0,C 180,E1 -12342.134,E2 -12342.134} C_VEL
LIN {X 0,Y 376.996,Z 525.534,A -85,B 0,C 180,E1 -12344.025,E2 -12344.025} C_VEL
LIN {X 0,Y 378.116,Z 517.268,A -85,B 0,C 180,E1 -12345.635,E2 -12345.635} C_VEL
LIN {X 0,Y 379.498,Z 507.341,A -85,B 0,C 180,E1 -12347.235,E2 -12347.235} C_VEL
LIN {X 0,Y 381.066,Z 496.329,A -85,B 0,C 180,E1 -12348.689,E2 -12348.689} C_VEL
LIN {X 0,Y 382.622,Z 484.06,A -85,B 0,C 180,E1 -12350.004,E2 -12350.004} C_VEL
LIN {X 0,Y 383.947,Z 472.527,A -85,B 0,C 180,E1 -12351.005,E2 -12351.005} C_VEL
LIN {X 0,Y 385.22,Z 459.647,A -85,B 0,C 180,E1 -12351.892,E2 -12351.892} C_VEL
LIN {X 0,Y 386.453,Z 446.017,A -85,B 0,C 180,E1 -12352.592,E2 -12352.592} C_VEL
LIN {X 0,Y 387.325,Z 431.992,A -85,B 0,C 180,E1 -12353.102,E2 -12353.102} C_VEL
LIN {X 0,Y 387.927,Z 412.836,A -85,B 0,C 180,E1 -12353.521,E2 -12353.521} C_VEL
LIN {X 0,Y 389.68,Z 326.217,A -85,B 0,C 180,E1 -12355.175,E2 -12355.175} C_VEL
LIN {X 0,Y 385.331,Z 303.834,A -85,B 0,C 180,E1 -12356.001,E2 -12356.001} C_VEL
LIN {X 0,Y 382.268,Z 290.18,A -85,B 0,C 180,E1 -12356.556,E2 -12356.556} C_VEL
LIN {X 0,Y 382.019,Z 286.471,A -85,B 0,C 180,E1 -12357.381,E2 -12357.381} C_VEL
LIN {X 0,Y 380,Z 277.124,A -85,B 0,C 180,E1 -12359.627,E2 -12359.627} C_VEL
LIN {X 0,Y 377.308,Z 266.324,A -85,B 0,C 180,E1 -12362.378,E2 -12362.378} C_VEL
LIN {X 0,Y 375.966,Z 261.286,A -85,B 0,C 180,E1 -12363.746,E2 -12363.746} C_VEL
LIN {X 0,Y 375.954,Z 261.282,A -85,B 0,C 180,E1 -12366.74,E2 -12366.74} C_VEL
LIN {X 0,Y 375.994,Z 261.273,A -85,B 0,C 180,E1 -12369.97,E2 -12369.97} C_VEL
LIN {X 0,Y 375.988,Z 261.275,A -85,B 0,C 180,E1 -12373.197,E2 -12373.197} C_VEL
LIN {X 0,Y 375.936,Z 261.281,A -85,B 0,C 180,E1 -12376.809,E2 -12376.809} C_VEL
LIN {X 0,Y 375.96,Z 261.278,A -85,B 0,C 180,E1 -12380.536,E2 -12380.536} C_VEL
LIN {X 0,Y 375.961,Z 261.263,A -85,B 0,C 180,E1 -12383.494,E2 -12383.494} C_VEL
LIN {X 0,Y 375.957,Z 261.269,A -85,B 0,C 180,E1 -12385.887,E2 -12385.887} C_VEL
LIN {X 0,Y 375.965,Z 261.273,A -85,B 0,C 180,E1 -12389.686,E2 -12389.686} C_VEL
LIN {X 0,Y 375.998,Z 261.269,A -85,B 0,C 180,E1 -12392.14,E2 -12392.14} C_VEL
LIN {X 0,Y 376.002,Z 261.272,A -85,B 0,C 180,E1 -12394.537,E2 -12394.537} C_VEL
LIN {X 0,Y 375.958,Z 261.28,A -85,B 0,C 180,E1 -12398.044,E2 -12398.044} C_VEL
LIN {X 0,Y 376.018,Z 261.271,A -85,B 0,C 180,E1 -12401.472,E2 -12401.472} C_VEL
LIN {X 0,Y 376.052,Z 261.261,A -85,B 0,C 180,E1 -12404.831,E2 -12404.831} C_VEL
LIN {X 0,Y 376.043,Z 261.259,A -85,B 0,C 180,E1 -12408.135,E2 -12408.135} C_VEL
LIN {X 0,Y 376.212,Z 261.239,A -85,B 0,C 180,E1 -12411.917,E2 -12411.917} C_VEL
LIN {X 0,Y 376.163,Z 261.252,A -85,B 0,C 180,E1 -12414.638,E2 -12414.638} C_VEL
LIN {X 0,Y 376.346,Z 261.229,A -85,B 0,C 180,E1 -12417.858,E2 -12417.858} C_VEL
LIN {X 0,Y 376.482,Z 261.21,A -85,B 0,C 180,E1 -12419.999,E2 -12419.999} C_VEL
LIN {X 0,Y 376.181,Z 261.253,A -85,B 0,C 180,E1 -12423.211,E2 -12423.211} C_VEL
LIN {X 0,Y 376.215,Z 261.241,A -85,B 0,C 180,E1 -12426.64,E2 -12426.64} C_VEL
LIN {X 0,Y 376.109,Z 261.252,A -85,B 0,C 180,E1 -12429.68,E2 -12429.68} C_VEL
LIN {X 0,Y 376.079,Z 261.257,A -85,B 0,C 180,E1 -12433.656,E2 -12433.656} C_VEL
LIN {X 0,Y 376.034,Z 261.265,A -85,B 0,C 180,E1 -12437.606,E2 -12437.606} C_VEL
LIN {X 0,Y 375.995,Z 261.271,A -85,B 0,C 180,E1 -12440.842,E2 -12440.842} C_VEL
LIN {X 0,Y 375.986,Z 261.271,A -85,B 0,C 180,E1 -12444.28,E2 -12444.28} C_VEL
LIN {X 0,Y 376.007,Z 261.271,A -85,B 0,C 180,E1 -12446.651,E2 -12446.651} C_VEL
LIN {X 0,Y 375.964,Z 261.274,A -85,B 0,C 180,E1 -12449.078,E2 -12449.078} C_VEL
LIN {X 0,Y 375.936,Z 261.284,A -85,B 0,C 180,E1 -12452.828,E2 -12452.828} C_VEL
LIN {X 0,Y 375.945,Z 261.268,A -85,B 0,C 180,E1 -12455.415,E2 -12455.415} C_VEL
LIN {X 0,Y 375.964,Z 261.273,A -85,B 0,C 180,E1 -12458.27,E2 -12458.27} C_VEL
LIN {X 0,Y 375.976,Z 261.273,A -85,B 0,C 180,E1 -12461.609,E2 -12461.609} C_VEL
LIN {X 0,Y 376.002,Z 261.274,A -85,B 0,C 180,E1 -12465.254,E2 -12465.254} C_VEL
LIN {X 0,Y 376.037,Z 261.379,A -85,B 0,C 180,E1 -12466.096,E2 -12466.096} C_VEL
LIN {X 0,Y 378.703,Z 272.287,A -85,B 0,C 180,E1 -12469.176,E2 -12469.176} C_VEL
LIN {X 0,Y 388.165,Z 293.158,A -85,B 0,C 180,E1 -12470.443,E2 -12470.443} C_VEL
LIN {X 0,Y 390.126,Z 300.999,A -85,B 0,C 180,E1 -12470.768,E2 -12470.768} C_VEL
LIN {X 0,Y 389.873,Z 323.095,A -85,B 0,C 180,E1 -12471.208,E2 -12471.208} C_VEL
LIN {X 0,Y 387.825,Z 408.823,A -85,B 0,C 180,E1 -12472.851,E2 -12472.851} C_VEL
LIN {X 0,Y 387.12,Z 422.796,A -85,B 0,C 180,E1 -12473.317,E2 -12473.317} C_VEL
LIN {X 0,Y 386.09,Z 436.382,A -85,B 0,C 180,E1 -12473.973,E2 -12473.973} C_VEL
LIN {X 0,Y 384.921,Z 450.299,A -85,B 0,C 180,E1 -12474.893,E2 -12474.893} C_VEL
LIN {X 0,Y 383.667,Z 462.029,A -85,B 0,C 180,E1 -12475.877,E2 -12475.877} C_VEL
LIN {X 0,Y 382.312,Z 472.992,A -85,B 0,C 180,E1 -12477.004,E2 -12477.004} C_VEL
LIN {X 0,Y 380.818,Z 484.037,A -85,B 0,C 180,E1 -12478.388,E2 -12478.388} C_VEL
LIN {X 0,Y 379.331,Z 494.459,A -85,B 0,C 180,E1 -12479.985,E2 -12479.985} C_VEL
LIN {X 0,Y 378.046,Z 503.611,A -85,B 0,C 180,E1 -12481.703,E2 -12481.703} C_VEL
LIN {X 0,Y 377.007,Z 511.32,A -85,B 0,C 180,E1 -12483.477,E2 -12483.477} C_VEL
LIN {X 0,Y 376.189,Z 517.24,A -85,B 0,C 180,E1 -12485.144,E2 -12485.144} C_VEL
LIN {X 0,Y 375.529,Z 522.208,A -85,B 0,C 180,E1 -12486.859,E2 -12486.859} C_VEL
LIN {X 0,Y 375.074,Z 526.159,A -85,B 0,C 180,E1 -12488.569,E2 -12488.569} C_VEL
LIN {X 0,Y 374.74,Z 529.17,A -85,B 0,C 180,E1 -12490.271,E2 -12490.271} C_VEL
LIN {X 0,Y 374.469,Z 531.787,A -85,B 0,C 180,E1 -12492.526,E2 -12492.526} C_VEL
LIN {X 0,Y 374.322,Z 532.939,A -85,B 0,C 180,E1 -12494.761,E2 -12494.761} C_VEL
LIN {X 0,Y 374.357,Z 532.69,A -85,B 0,C 180,E1 -12496.981,E2 -12496.981} C_VEL
LIN {X 0,Y 374.429,Z 532.046,A -85,B 0,C 180,E1 -12498.085,E2 -12498.085} C_VEL
LIN {X 0,Y 374.451,Z 529.735,A -85,B 0,C 180,E1 -12500.275,E2 -12500.275} C_VEL
LIN {X 0,Y 374.803,Z 525.994,A -85,B 0,C 180,E1 -12502.458,E2 -12502.458} C_VEL
LIN {X 0,Y 375.137,Z 520.751,A -85,B 0,C 180,E1 -12504.625,E2 -12504.625} C_VEL
LIN {X 0,Y 375.564,Z 515.669,A -85,B 0,C 180,E1 -12506.245,E2 -12506.245} C_VEL
LIN {X 0,Y 376.196,Z 508.438,A -85,B 0,C 180,E1 -12508.127,E2 -12508.127} C_VEL
LIN {X 0,Y 376.987,Z 500.864,A -85,B 0,C 180,E1 -12509.733,E2 -12509.733} C_VEL
LIN {X 0,Y 378.046,Z 491.768,A -85,B 0,C 180,E1 -12511.332,E2 -12511.332} C_VEL
LIN {X 0,Y 379.231,Z 480.768,A -85,B 0,C 180,E1 -12512.921,E2 -12512.921} C_VEL
LIN {X 0,Y 380.404,Z 469.545,A -85,B 0,C 180,E1 -12514.238,E2 -12514.238} C_VEL
LIN {X 0,Y 381.526,Z 457.174,A -85,B 0,C 180,E1 -12515.417,E2 -12515.417} C_VEL
LIN {X 0,Y 382.521,Z 445.245,A -85,B 0,C 180,E1 -12516.329,E2 -12516.329} C_VEL
LIN {X 0,Y 383.339,Z 431.867,A -85,B 0,C 180,E1 -12517.129,E2 -12517.129} C_VEL
LIN {X 0,Y 383.165,Z 426.296,A -85,B 0,C 180,E1 -12517.423,E2 -12517.423} C_VEL
LIN {X 0,Y 380.792,Z 417.248,A -85,B 0,C 180,E1 -12517.926,E2 -12517.926} C_VEL
LIN {X 0,Y 378.31,Z 408.07,A -85,B 0,C 180,E1 -12518.356,E2 -12518.356} C_VEL
LIN {X 0,Y 377.832,Z 402.297,A -85,B 0,C 180,E1 -12518.519,E2 -12518.519} C_VEL
LIN {X 0,Y 379.759,Z 301.325,A -85,B 0,C 180,E1 -12520.433,E2 -12520.433} C_VEL
LIN {X 0,Y 376.535,Z 286.681,A -85,B 0,C 180,E1 -12520.92,E2 -12520.92} C_VEL
LIN {X 0,Y 371.083,Z 271.81,A -85,B 0,C 180,E1 -12521.586,E2 -12521.586} C_VEL
LIN {X 0,Y 369.013,Z 262.15,A -85,B 0,C 180,E1 -12524.086,E2 -12524.086} C_VEL
LIN {X 0,Y 368.988,Z 262.15,A -85,B 0,C 180,E1 -12527.769,E2 -12527.769} C_VEL
LIN {X 0,Y 368.928,Z 262.153,A -85,B 0,C 180,E1 -12531.219,E2 -12531.219} C_VEL
LIN {X 0,Y 368.945,Z 262.149,A -85,B 0,C 180,E1 -12534.776,E2 -12534.776} C_VEL
LIN {X 0,Y 368.975,Z 262.145,A -85,B 0,C 180,E1 -12538.436,E2 -12538.436} C_VEL
LIN {X 0,Y 368.888,Z 262.157,A -85,B 0,C 180,E1 -12542.238,E2 -12542.238} C_VEL
LIN {X 0,Y 368.916,Z 262.154,A -85,B 0,C 180,E1 -12545.002,E2 -12545.002} C_VEL
LIN {X 0,Y 368.9,Z 262.155,A -85,B 0,C 180,E1 -12548.642,E2 -12548.642} C_VEL
LIN {X 0,Y 368.929,Z 262.152,A -85,B 0,C 180,E1 -12552.021,E2 -12552.021} C_VEL
LIN {X 0,Y 368.977,Z 262.15,A -85,B 0,C 180,E1 -12555.194,E2 -12555.194} C_VEL
LIN {X 0,Y 368.929,Z 262.151,A -85,B 0,C 180,E1 -12558.187,E2 -12558.187} C_VEL
LIN {X 0,Y 368.902,Z 262.159,A -85,B 0,C 180,E1 -12561.36,E2 -12561.36} C_VEL
LIN {X 0,Y 368.925,Z 262.158,A -85,B 0,C 180,E1 -12565.148,E2 -12565.148} C_VEL
LIN {X 0,Y 368.918,Z 262.159,A -85,B 0,C 180,E1 -12569.048,E2 -12569.048} C_VEL
LIN {X 0,Y 368.976,Z 262.146,A -85,B 0,C 180,E1 -12571.566,E2 -12571.566} C_VEL
LIN {X 0,Y 368.947,Z 262.152,A -85,B 0,C 180,E1 -12575.226,E2 -12575.226} C_VEL
LIN {X 0,Y 368.927,Z 262.157,A -85,B 0,C 180,E1 -12578.975,E2 -12578.975} C_VEL
LIN {X 0,Y 368.981,Z 262.146,A -85,B 0,C 180,E1 -12582.259,E2 -12582.259} C_VEL
LIN {X 0,Y 369.028,Z 262.14,A -85,B 0,C 180,E1 -12586.229,E2 -12586.229} C_VEL
LIN {X 0,Y 369.059,Z 262.136,A -85,B 0,C 180,E1 -12590.133,E2 -12590.133} C_VEL
LIN {X 0,Y 369.194,Z 262.118,A -85,B 0,C 180,E1 -12593.443,E2 -12593.443} C_VEL
LIN {X 0,Y 369.312,Z 262.104,A -85,B 0,C 180,E1 -12597.82,E2 -12597.82} C_VEL
LIN {X 0,Y 369.451,Z 262.088,A -85,B 0,C 180,E1 -12600.001,E2 -12600.001} C_VEL
LIN {X 0,Y 369.312,Z 262.107,A -85,B 0,C 180,E1 -12602.183,E2 -12602.183} C_VEL
LIN {X 0,Y 369.195,Z 262.122,A -85,B 0,C 180,E1 -12606.56,E2 -12606.56} C_VEL
LIN {X 0,Y 369.062,Z 262.137,A -85,B 0,C 180,E1 -12609.87,E2 -12609.87} C_VEL
LIN {X 0,Y 369.032,Z 262.14,A -85,B 0,C 180,E1 -12613.774,E2 -12613.774} C_VEL
LIN {X 0,Y 368.998,Z 262.145,A -85,B 0,C 180,E1 -12617.77,E2 -12617.77} C_VEL
LIN {X 0,Y 368.906,Z 262.154,A -85,B 0,C 180,E1 -12621.222,E2 -12621.222} C_VEL
LIN {X 0,Y 368.952,Z 262.149,A -85,B 0,C 180,E1 -12624.777,E2 -12624.777} C_VEL
LIN {X 0,Y 368.969,Z 262.146,A -85,B 0,C 180,E1 -12627.204,E2 -12627.204} C_VEL
LIN {X 0,Y 368.922,Z 262.156,A -85,B 0,C 180,E1 -12629.691,E2 -12629.691} C_VEL
LIN {X 0,Y 368.898,Z 262.158,A -85,B 0,C 180,E1 -12633.539,E2 -12633.539} C_VEL
LIN {X 0,Y 368.902,Z 262.154,A -85,B 0,C 180,E1 -12636.857,E2 -12636.857} C_VEL
LIN {X 0,Y 368.911,Z 262.154,A -85,B 0,C 180,E1 -12640.371,E2 -12640.371} C_VEL
LIN {X 0,Y 368.883,Z 262.162,A -85,B 0,C 180,E1 -12643.617,E2 -12643.617} C_VEL
LIN {X 0,Y 368.886,Z 262.156,A -85,B 0,C 180,E1 -12646.697,E2 -12646.697} C_VEL
LIN {X 0,Y 368.912,Z 262.159,A -85,B 0,C 180,E1 -12649.644,E2 -12649.644} C_VEL
LIN {X 0,Y 368.902,Z 262.157,A -85,B 0,C 180,E1 -12653.146,E2 -12653.146} C_VEL
LIN {X 0,Y 368.899,Z 262.16,A -85,B 0,C 180,E1 -12656.463,E2 -12656.463} C_VEL
LIN {X 0,Y 368.958,Z 262.3,A -85,B 0,C 180,E1 -12658.314,E2 -12658.314} C_VEL
LIN {X 0,Y 372.036,Z 276.118,A -85,B 0,C 180,E1 -12661.512,E2 -12661.512} C_VEL
LIN {X 0,Y 373.731,Z 284.956,A -85,B 0,C 180,E1 -12663.474,E2 -12663.474} C_VEL
LIN {X 0,Y 373.334,Z 290.399,A -85,B 0,C 180,E1 -12664.58,E2 -12664.58} C_VEL
LIN {X 0,Y 379.426,Z 327.427,A -85,B 0,C 180,E1 -12665.703,E2 -12665.703} C_VEL
LIN {X 0,Y 377.535,Z 428.23,A -85,B 0,C 180,E1 -12667.639,E2 -12667.639} C_VEL
LIN {X 0,Y 376.839,Z 443.036,A -85,B 0,C 180,E1 -12668.136,E2 -12668.136} C_VEL
LIN {X 0,Y 375.817,Z 457.108,A -85,B 0,C 180,E1 -12668.829,E2 -12668.829} C_VEL
LIN {X 0,Y 374.901,Z 469.74,A -85,B 0,C 180,E1 -12669.67,E2 -12669.67} C_VEL
LIN {X 0,Y 373.612,Z 482.894,A -85,B 0,C 180,E1 -12670.781,E2 -12670.781} C_VEL
LIN {X 0,Y 372.383,Z 494.455,A -85,B 0,C 180,E1 -12671.999,E2 -12671.999} C_VEL
LIN {X 0,Y 371.299,Z 504.072,A -85,B 0,C 180,E1 -12673.223,E2 -12673.223} C_VEL
LIN {X 0,Y 370.155,Z 514.772,A -85,B 0,C 180,E1 -12674.867,E2 -12674.867} C_VEL
LIN {X 0,Y 369.375,Z 523.815,A -85,B 0,C 180,E1 -12676.566,E2 -12676.566} C_VEL
LIN {X 0,Y 368.516,Z 532.035,A -85,B 0,C 180,E1 -12678.449,E2 -12678.449} C_VEL
LIN {X 0,Y 367.993,Z 537.899,A -85,B 0,C 180,E1 -12680.103,E2 -12680.103} C_VEL
LIN {X 0,Y 367.706,Z 542.72,A -85,B 0,C 180,E1 -12681.758,E2 -12681.758} C_VEL
LIN {X 0,Y 367.488,Z 547.722,A -85,B 0,C 180,E1 -12683.978,E2 -12683.978} C_VEL
LIN {X 0,Y 367.412,Z 550.408,A -85,B 0,C 180,E1 -12685.612,E2 -12685.612} C_VEL
LIN {X 0,Y 367.37,Z 552.773,A -85,B 0,C 180,E1 -12687.807,E2 -12687.807} C_VEL
LIN {X 0,Y 367.457,Z 553.777,A -85,B 0,C 180,E1 -12690,E2 -12690} C_VEL
LIN {X 0,Y 367.354,Z 553.437,A -85,B 0,C 180,E1 -12692.193,E2 -12692.193} C_VEL
LIN {X 0,Y 367.415,Z 551.768,A -85,B 0,C 180,E1 -12694.388,E2 -12694.388} C_VEL
LIN {X 0,Y 367.555,Z 548.736,A -85,B 0,C 180,E1 -12696.588,E2 -12696.588} C_VEL
LIN {X 0,Y 367.862,Z 544.265,A -85,B 0,C 180,E1 -12698.791,E2 -12698.791} C_VEL
LIN {X 0,Y 368.258,Z 539.854,A -85,B 0,C 180,E1 -12700.445,E2 -12700.445} C_VEL
LIN {X 0,Y 369.136,Z 533.496,A -85,B 0,C 180,E1 -12702.368,E2 -12702.368} C_VEL
LIN {X 0,Y 370.065,Z 525.619,A -85,B 0,C 180,E1 -12704.293,E2 -12704.293} C_VEL
LIN {X 0,Y 371.255,Z 517.411,A -85,B 0,C 180,E1 -12705.931,E2 -12705.931} C_VEL
LIN {X 0,Y 372.706,Z 507.553,A -85,B 0,C 180,E1 -12707.56,E2 -12707.56} C_VEL
LIN {X 0,Y 374.358,Z 496.622,A -85,B 0,C 180,E1 -12709.037,E2 -12709.037} C_VEL
LIN {X 0,Y 375.968,Z 484.519,A -85,B 0,C 180,E1 -12710.374,E2 -12710.374} C_VEL
LIN {X 0,Y 377.508,Z 471.975,A -85,B 0,C 180,E1 -12711.479,E2 -12711.479} C_VEL
LIN {X 0,Y 378.917,Z 458.301,A -85,B 0,C 180,E1 -12712.419,E2 -12712.419} C_VEL
LIN {X 0,Y 380.158,Z 444.302,A -85,B 0,C 180,E1 -12713.131,E2 -12713.131} C_VEL
LIN {X 0,Y 381.075,Z 430.659,A -85,B 0,C 180,E1 -12713.612,E2 -12713.612} C_VEL
LIN {X 0,Y 381.707,Z 409.293,A -85,B 0,C 180,E1 -12714.071,E2 -12714.071} C_VEL
LIN {X 0,Y 383.457,Z 327.287,A -85,B 0,C 180,E1 -12715.661,E2 -12715.661} C_VEL
LIN {X 0,Y 378.858,Z 303.783,A -85,B 0,C 180,E1 -12716.556,E2 -12716.556} C_VEL
LIN {X 0,Y 375.548,Z 289.905,A -85,B 0,C 180,E1 -12717.168,E2 -12717.168} C_VEL
LIN {X 0,Y 373.366,Z 279.583,A -85,B 0,C 180,E1 -12719.691,E2 -12719.691} C_VEL
LIN {X 0,Y 370.812,Z 269.332,A -85,B 0,C 180,E1 -12722.35,E2 -12722.35} C_VEL
LIN {X 0,Y 368.927,Z 262.157,A -85,B 0,C 180,E1 -12724.356,E2 -12724.356} C_VEL
LIN {X 0,Y 368.904,Z 262.155,A -85,B 0,C 180,E1 -12727.562,E2 -12727.562} C_VEL
LIN {X 0,Y 368.953,Z 262.146,A -85,B 0,C 180,E1 -12730.363,E2 -12730.363} C_VEL
LIN {X 0,Y 368.93,Z 262.154,A -85,B 0,C 180,E1 -12733.622,E2 -12733.622} C_VEL
LIN {X 0,Y 368.888,Z 262.16,A -85,B 0,C 180,E1 -12736.695,E2 -12736.695} C_VEL
LIN {X 0,Y 368.91,Z 262.157,A -85,B 0,C 180,E1 -12739.642,E2 -12739.642} C_VEL
LIN {X 0,Y 368.899,Z 262.147,A -85,B 0,C 180,E1 -12743.143,E2 -12743.143} C_VEL
LIN {X 0,Y 368.894,Z 262.158,A -85,B 0,C 180,E1 -12746.46,E2 -12746.46} C_VEL
LIN {X 0,Y 368.92,Z 262.156,A -85,B 0,C 180,E1 -12750.309,E2 -12750.309} C_VEL
LIN {X 0,Y 368.978,Z 262.146,A -85,B 0,C 180,E1 -12753.534,E2 -12753.534} C_VEL
LIN {X 0,Y 368.962,Z 262.146,A -85,B 0,C 180,E1 -12756.42,E2 -12756.42} C_VEL
LIN {X 0,Y 368.931,Z 262.148,A -85,B 0,C 180,E1 -12759.945,E2 -12759.945} C_VEL
LIN {X 0,Y 368.97,Z 262.145,A -85,B 0,C 180,E1 -12763.397,E2 -12763.397} C_VEL
LIN {X 0,Y 369.051,Z 262.138,A -85,B 0,C 180,E1 -12766.789,E2 -12766.789} C_VEL
LIN {X 0,Y 369.061,Z 262.138,A -85,B 0,C 180,E1 -12770.13,E2 -12770.13} C_VEL
LIN {X 0,Y 369.155,Z 262.116,A -85,B 0,C 180,E1 -12772.34,E2 -12772.34} C_VEL
LIN {X 0,Y 369.136,Z 262.127,A -85,B 0,C 180,E1 -12774.536,E2 -12774.536} C_VEL
LIN {X 0,Y 369.311,Z 262.104,A -85,B 0,C 180,E1 -12777.817,E2 -12777.817} C_VEL
LIN {X 0,Y 369.451,Z 262.086,A -85,B 0,C 180,E1 -12779.999,E2 -12779.999} C_VEL
LIN {X 0,Y 369.31,Z 262.102,A -85,B 0,C 180,E1 -12782.18,E2 -12782.18} C_VEL
LIN {X 0,Y 369.185,Z 262.117,A -85,B 0,C 180,E1 -12786.625,E2 -12786.625} C_VEL
LIN {X 0,Y 369.112,Z 262.131,A -85,B 0,C 180,E1 -12788.76,E2 -12788.76} C_VEL
LIN {X 0,Y 368.995,Z 262.145,A -85,B 0,C 180,E1 -12792.092,E2 -12792.092} C_VEL
LIN {X 0,Y 368.987,Z 262.147,A -85,B 0,C 180,E1 -12795.464,E2 -12795.464} C_VEL
LIN {X 0,Y 368.979,Z 262.151,A -85,B 0,C 180,E1 -12798.891,E2 -12798.891} C_VEL
LIN {X 0,Y 368.935,Z 262.154,A -85,B 0,C 180,E1 -12802.393,E2 -12802.393} C_VEL
LIN {X 0,Y 368.988,Z 262.147,A -85,B 0,C 180,E1 -12805.979,E2 -12805.979} C_VEL
LIN {X 0,Y 368.955,Z 262.15,A -85,B 0,C 180,E1 -12808.812,E2 -12808.812} C_VEL
LIN {X 0,Y 368.886,Z 262.155,A -85,B 0,C 180,E1 -12812.237,E2 -12812.237} C_VEL
LIN {X 0,Y 368.916,Z 262.143,A -85,B 0,C 180,E1 -12815.001,E2 -12815.001} C_VEL
LIN {X 0,Y 368.899,Z 262.15,A -85,B 0,C 180,E1 -12818.64,E2 -12818.64} C_VEL
LIN {X 0,Y 368.928,Z 262.149,A -85,B 0,C 180,E1 -12822.019,E2 -12822.019} C_VEL
LIN {X 0,Y 369.004,Z 262.322,A -85,B 0,C 180,E1 -12825.55,E2 -12825.55} C_VEL
LIN {X 0,Y 371.502,Z 272.47,A -85,B 0,C 180,E1 -12828.501,E2 -12828.501} C_VEL
LIN {X 0,Y 379.522,Z 289.475,A -85,B 0,C 180,E1 -12829.624,E2 -12829.624} C_VEL
LIN {X 0,Y 382.912,Z 297.674,A -85,B 0,C 180,E1 -12830.095,E2 -12830.095} C_VEL
LIN {X 0,Y 384.064,Z 302.971,A -85,B 0,C 180,E1 -12830.306,E2 -12830.306} C_VEL
LIN {X 0,Y 381.516,Z 409.278,A -85,B 0,C 180,E1 -12832.38,E2 -12832.38} C_VEL
LIN {X 0,Y 380.772,Z 423.16,A -85,B 0,C 180,E1 -12832.852,E2 -12832.852} C_VEL
LIN {X 0,Y 379.686,Z 436.682,A -85,B 0,C 180,E1 -12833.515,E2 -12833.515} C_VEL
LIN {X 0,Y 378.566,Z 449.618,A -85,B 0,C 180,E1 -12834.377,E2 -12834.377} C_VEL
LIN {X 0,Y 377.168,Z 461.972,A -85,B 0,C 180,E1 -12835.418,E2 -12835.418} C_VEL
LIN {X 0,Y 375.811,Z 472.588,A -85,B 0,C 180,E1 -12836.519,E2 -12836.519} C_VEL
LIN {X 0,Y 374.267,Z 483.458,A -85,B 0,C 180,E1 -12837.887,E2 -12837.887} C_VEL
LIN {X 0,Y 372.799,Z 493.373,A -85,B 0,C 180,E1 -12839.403,E2 -12839.403} C_VEL
LIN {X 0,Y 371.405,Z 502.743,A -85,B 0,C 180,E1 -12841.15,E2 -12841.15} C_VEL
LIN {X 0,Y 370.254,Z 510.43,A -85,B 0,C 180,E1 -12842.9,E2 -12842.9} C_VEL
LIN {X 0,Y 369.335,Z 516.73,A -85,B 0,C 180,E1 -12844.651,E2 -12844.651} C_VEL
LIN {X 0,Y 368.617,Z 521.854,A -85,B 0,C 180,E1 -12846.399,E2 -12846.399} C_VEL
LIN {X 0,Y 368.102,Z 525.945,A -85,B 0,C 180,E1 -12848.143,E2 -12848.143} C_VEL
LIN {X 0,Y 367.724,Z 529.024,A -85,B 0,C 180,E1 -12849.879,E2 -12849.879} C_VEL
LIN {X 0,Y 367.404,Z 531.809,A -85,B 0,C 180,E1 -12852.179,E2 -12852.179} C_VEL
LIN {X 0,Y 367.237,Z 533.11,A -85,B 0,C 180,E1 -12854.46,E2 -12854.46} C_VEL
LIN {X 0,Y 367.241,Z 532.986,A -85,B 0,C 180,E1 -12856.724,E2 -12856.724} C_VEL
LIN {X 0,Y 367.335,Z 532.402,A -85,B 0,C 180,E1 -12857.851,E2 -12857.851} C_VEL
LIN {X 0,Y 367.338,Z 530.215,A -85,B 0,C 180,E1 -12860.085,E2 -12860.085} C_VEL
LIN {X 0,Y 367.675,Z 526.601,A -85,B 0,C 180,E1 -12862.311,E2 -12862.311} C_VEL
LIN {X 0,Y 367.972,Z 522.515,A -85,B 0,C 180,E1 -12864.127,E2 -12864.127} C_VEL
LIN {X 0,Y 368.45,Z 516.549,A -85,B 0,C 180,E1 -12866.172,E2 -12866.172} C_VEL
LIN {X 0,Y 369.095,Z 509.47,A -85,B 0,C 180,E1 -12868.091,E2 -12868.091} C_VEL
LIN {X 0,Y 369.898,Z 502.066,A -85,B 0,C 180,E1 -12869.728,E2 -12869.728} C_VEL
LIN {X 0,Y 370.958,Z 493.169,A -85,B 0,C 180,E1 -12871.357,E2 -12871.357} C_VEL
LIN {X 0,Y 372.156,Z 482.423,A -85,B 0,C 180,E1 -12872.977,E2 -12872.977} C_VEL
LIN {X 0,Y 373.364,Z 471.531,A -85,B 0,C 180,E1 -12874.318,E2 -12874.318} C_VEL
LIN {X 0,Y 374.557,Z 459.478,A -85,B 0,C 180,E1 -12875.532,E2 -12875.532} C_VEL
LIN {X 0,Y 375.682,Z 446.387,A -85,B 0,C 180,E1 -12876.58,E2 -12876.58} C_VEL
LIN {X 0,Y 376.508,Z 433.685,A -85,B 0,C 180,E1 -12877.373,E2 -12877.373} C_VEL
LIN {X 0,Y 377.259,Z 419.262,A -85,B 0,C 180,E1 -12878.031,E2 -12878.031} C_VEL
LIN {X 0,Y 377.775,Z 404.987,A -85,B 0,C 180,E1 -12878.458,E2 -12878.458} C_VEL
LIN {X 0,Y 377.832,Z 402.297,A -85,B 0,C 180,E1 -12878.519,E2 -12878.519} C_VEL
LIN {X 0,Y 377.422,Z 396.496,A -85,B 0,C 180,E1 -12878.671,E2 -12878.671} C_VEL
LIN {X 0,Y 372.295,Z 377.79,A -85,B 0,C 180,E1 -12879.319,E2 -12879.319} C_VEL
LIN {X 0,Y 371.751,Z 371.974,A -85,B 0,C 180,E1 -12879.465,E2 -12879.465} C_VEL
LIN {X 0,Y 373.169,Z 302.532,A -85,B 0,C 180,E1 -12880.8,E2 -12880.8} C_VEL
LIN {X 0,Y 370.158,Z 288.893,A -85,B 0,C 180,E1 -12881.264,E2 -12881.264} C_VEL
LIN {X 0,Y 363.939,Z 272.113,A -85,B 0,C 180,E1 -12882.012,E2 -12882.012} C_VEL
LIN {X 0,Y 361.964,Z 263.032,A -85,B 0,C 180,E1 -12884.393,E2 -12884.393} C_VEL
LIN {X 0,Y 361.948,Z 263.024,A -85,B 0,C 180,E1 -12888.1,E2 -12888.1} C_VEL
LIN {X 0,Y 361.886,Z 263.034,A -85,B 0,C 180,E1 -12891.653,E2 -12891.653} C_VEL
LIN {X 0,Y 361.915,Z 263.027,A -85,B 0,C 180,E1 -12895.291,E2 -12895.291} C_VEL
LIN {X 0,Y 361.91,Z 263.03,A -85,B 0,C 180,E1 -12897.778,E2 -12897.778} C_VEL
LIN {X 0,Y 361.834,Z 263.038,A -85,B 0,C 180,E1 -12901.286,E2 -12901.286} C_VEL
LIN {X 0,Y 361.841,Z 263.034,A -85,B 0,C 180,E1 -12904.281,E2 -12904.281} C_VEL
LIN {X 0,Y 361.859,Z 263.036,A -85,B 0,C 180,E1 -12907.225,E2 -12907.225} C_VEL
LIN {X 0,Y 361.893,Z 263.028,A -85,B 0,C 180,E1 -12910.769,E2 -12910.769} C_VEL
LIN {X 0,Y 361.921,Z 263.024,A -85,B 0,C 180,E1 -12914.351,E2 -12914.351} C_VEL
LIN {X 0,Y 361.874,Z 263.033,A -85,B 0,C 180,E1 -12917.56,E2 -12917.56} C_VEL
LIN {X 0,Y 361.863,Z 263.035,A -85,B 0,C 180,E1 -12920.973,E2 -12920.973} C_VEL
LIN {X 0,Y 361.863,Z 263.033,A -85,B 0,C 180,E1 -12924.656,E2 -12924.656} C_VEL
LIN {X 0,Y 361.826,Z 263.036,A -85,B 0,C 180,E1 -12928.372,E2 -12928.372} C_VEL
LIN {X 0,Y 361.892,Z 263.033,A -85,B 0,C 180,E1 -12930.957,E2 -12930.957} C_VEL
LIN {X 0,Y 361.944,Z 263.023,A -85,B 0,C 180,E1 -12933.476,E2 -12933.476} C_VEL
LIN {X 0,Y 361.88,Z 263.033,A -85,B 0,C 180,E1 -12937.146,E2 -12937.146} C_VEL
LIN {X 0,Y 361.896,Z 263.032,A -85,B 0,C 180,E1 -12940.725,E2 -12940.725} C_VEL
LIN {X 0,Y 361.923,Z 263.027,A -85,B 0,C 180,E1 -12943.067,E2 -12943.067} C_VEL
LIN {X 0,Y 361.99,Z 263.02,A -85,B 0,C 180,E1 -12946.529,E2 -12946.529} C_VEL
LIN {X 0,Y 362.023,Z 263.012,A -85,B 0,C 180,E1 -12949.939,E2 -12949.939} C_VEL
LIN {X 0,Y 362.156,Z 262.995,A -85,B 0,C 180,E1 -12953.315,E2 -12953.315} C_VEL
LIN {X 0,Y 362.276,Z 262.98,A -85,B 0,C 180,E1 -12957.778,E2 -12957.778} C_VEL
LIN {X 0,Y 362.421,Z 262.963,A -85,B 0,C 180,E1 -12960.001,E2 -12960.001} C_VEL
LIN {X 0,Y 362.276,Z 262.984,A -85,B 0,C 180,E1 -12962.225,E2 -12962.225} C_VEL
LIN {X 0,Y 362.157,Z 262.998,A -85,B 0,C 180,E1 -12966.688,E2 -12966.688} C_VEL
LIN {X 0,Y 362.026,Z 263.015,A -85,B 0,C 180,E1 -12970.064,E2 -12970.064} C_VEL
LIN {X 0,Y 361.993,Z 263.018,A -85,B 0,C 180,E1 -12973.9,E2 -12973.9} C_VEL
LIN {X 0,Y 361.964,Z 263.023,A -85,B 0,C 180,E1 -12977.94,E2 -12977.94} C_VEL
LIN {X 0,Y 361.858,Z 263.034,A -85,B 0,C 180,E1 -12981.656,E2 -12981.656} C_VEL
LIN {X 0,Y 361.924,Z 263.024,A -85,B 0,C 180,E1 -12985.292,E2 -12985.292} C_VEL
LIN {X 0,Y 361.92,Z 263.028,A -85,B 0,C 180,E1 -12987.779,E2 -12987.779} C_VEL
LIN {X 0,Y 361.858,Z 263.035,A -85,B 0,C 180,E1 -12991.629,E2 -12991.629} C_VEL
LIN {X 0,Y 361.874,Z 263.032,A -85,B 0,C 180,E1 -12995.346,E2 -12995.346} C_VEL
LIN {X 0,Y 361.87,Z 263.031,A -85,B 0,C 180,E1 -12999.028,E2 -12999.028} C_VEL
LIN {X 0,Y 361.836,Z 263.035,A -85,B 0,C 180,E1 -13002.83,E2 -13002.83} C_VEL
LIN {X 0,Y 361.819,Z 263.04,A -85,B 0,C 180,E1 -13005.948,E2 -13005.948} C_VEL
LIN {X 0,Y 361.836,Z 263.037,A -85,B 0,C 180,E1 -13009.246,E2 -13009.246} C_VEL
LIN {X 0,Y 361.864,Z 263.032,A -85,B 0,C 180,E1 -13012.779,E2 -13012.779} C_VEL
LIN {X 0,Y 361.856,Z 263.039,A -85,B 0,C 180,E1 -13015.721,E2 -13015.721} C_VEL
LIN {X 0,Y 361.917,Z 263.193,A -85,B 0,C 180,E1 -13017.97,E2 -13017.97} C_VEL
LIN {X 0,Y 364.971,Z 276.963,A -85,B 0,C 180,E1 -13021.223,E2 -13021.223} C_VEL
LIN {X 0,Y 366.772,Z 285.817,A -85,B 0,C 180,E1 -13023.237,E2 -13023.237} C_VEL
LIN {X 0,Y 366.561,Z 290.206,A -85,B 0,C 180,E1 -13024.155,E2 -13024.155} C_VEL
LIN {X 0,Y 372.759,Z 327.714,A -85,B 0,C 180,E1 -13025.323,E2 -13025.323} C_VEL
LIN {X 0,Y 370.838,Z 428.154,A -85,B 0,C 180,E1 -13027.286,E2 -13027.286} C_VEL
LIN {X 0,Y 370.104,Z 442.908,A -85,B 0,C 180,E1 -13027.79,E2 -13027.79} C_VEL
LIN {X 0,Y 369.07,Z 456.966,A -85,B 0,C 180,E1 -13028.496,E2 -13028.496} C_VEL
LIN {X 0,Y 368.037,Z 470.315,A -85,B 0,C 180,E1 -13029.407,E2 -13029.407} C_VEL
LIN {X 0,Y 366.695,Z 483.449,A -85,B 0,C 180,E1 -13030.549,E2 -13030.549} C_VEL
LIN {X 0,Y 365.44,Z 494.879,A -85,B 0,C 180,E1 -13031.79,E2 -13031.79} C_VEL
LIN {X 0,Y 364.2,Z 505.377,A -85,B 0,C 180,E1 -13033.175,E2 -13033.175} C_VEL
LIN {X 0,Y 363.07,Z 515.816,A -85,B 0,C 180,E1 -13034.852,E2 -13034.852} C_VEL
LIN {X 0,Y 362.294,Z 524.432,A -85,B 0,C 180,E1 -13036.539,E2 -13036.539} C_VEL
LIN {X 0,Y 361.398,Z 532.625,A -85,B 0,C 180,E1 -13038.502,E2 -13038.502} C_VEL
LIN {X 0,Y 360.835,Z 539.221,A -85,B 0,C 180,E1 -13040.471,E2 -13040.471} C_VEL
LIN {X 0,Y 360.493,Z 545.058,A -85,B 0,C 180,E1 -13042.72,E2 -13042.72} C_VEL
LIN {X 0,Y 360.346,Z 548.391,A -85,B 0,C 180,E1 -13044.404,E2 -13044.404} C_VEL
LIN {X 0,Y 360.286,Z 551.499,A -85,B 0,C 180,E1 -13046.645,E2 -13046.645} C_VEL
LIN {X 0,Y 360.32,Z 553.216,A -85,B 0,C 180,E1 -13048.882,E2 -13048.882} C_VEL
LIN {X 0,Y 360.36,Z 553.568,A -85,B 0,C 180,E1 -13050,E2 -13050} C_VEL
LIN {X 0,Y 360.259,Z 553.265,A -85,B 0,C 180,E1 -13052.236,E2 -13052.236} C_VEL
LIN {X 0,Y 360.327,Z 551.633,A -85,B 0,C 180,E1 -13054.474,E2 -13054.474} C_VEL
LIN {X 0,Y 360.486,Z 548.639,A -85,B 0,C 180,E1 -13056.717,E2 -13056.717} C_VEL
LIN {X 0,Y 360.811,Z 544.208,A -85,B 0,C 180,E1 -13058.964,E2 -13058.964} C_VEL
LIN {X 0,Y 361.419,Z 538.213,A -85,B 0,C 180,E1 -13061.213,E2 -13061.213} C_VEL
LIN {X 0,Y 362.472,Z 531.493,A -85,B 0,C 180,E1 -13063.168,E2 -13063.168} C_VEL
LIN {X 0,Y 363.544,Z 523.17,A -85,B 0,C 180,E1 -13065.127,E2 -13065.127} C_VEL
LIN {X 0,Y 364.874,Z 514.527,A -85,B 0,C 180,E1 -13066.793,E2 -13066.793} C_VEL
LIN {X 0,Y 366.524,Z 504.086,A -85,B 0,C 180,E1 -13068.444,E2 -13068.444} C_VEL
LIN {X 0,Y 368.3,Z 492.436,A -85,B 0,C 180,E1 -13069.943,E2 -13069.943} C_VEL
LIN {X 0,Y 369.915,Z 480.802,A -85,B 0,C 180,E1 -13071.16,E2 -13071.16} C_VEL
LIN {X 0,Y 371.46,Z 468.024,A -85,B 0,C 180,E1 -13072.234,E2 -13072.234} C_VEL
LIN {X 0,Y 372.858,Z 454.765,A -85,B 0,C 180,E1 -13073.097,E2 -13073.097} C_VEL
LIN {X 0,Y 374.087,Z 441.104,A -85,B 0,C 180,E1 -13073.749,E2 -13073.749} C_VEL
LIN {X 0,Y 374.933,Z 427.015,A -85,B 0,C 180,E1 -13074.207,E2 -13074.207} C_VEL
LIN {X 0,Y 377.257,Z 328.439,A -85,B 0,C 180,E1 -13076.161,E2 -13076.161} C_VEL
LIN {X 0,Y 372.667,Z 304.937,A -85,B 0,C 180,E1 -13077.086,E2 -13077.086} C_VEL
LIN {X 0,Y 369.855,Z 293.245,A -85,B 0,C 180,E1 -13077.609,E2 -13077.609} C_VEL
LIN {X 0,Y 368.349,Z 289.657,A -85,B 0,C 180,E1 -13077.845,E2 -13077.845} C_VEL
LIN {X 0,Y 365.643,Z 277.363,A -85,B 0,C 180,E1 -13080.969,E2 -13080.969} C_VEL
LIN {X 0,Y 362.515,Z 265.551,A -85,B 0,C 180,E1 -13084.208,E2 -13084.208} C_VEL
LIN {X 0,Y 361.908,Z 263.03,A -85,B 0,C 180,E1 -13084.949,E2 -13084.949} C_VEL
LIN {X 0,Y 361.869,Z 263.036,A -85,B 0,C 180,E1 -13088.423,E2 -13088.423} C_VEL
LIN {X 0,Y 361.873,Z 263.027,A -85,B 0,C 180,E1 -13091.323,E2 -13091.323} C_VEL
LIN {X 0,Y 361.903,Z 263.033,A -85,B 0,C 180,E1 -13094.354,E2 -13094.354} C_VEL
LIN {X 0,Y 361.836,Z 263.037,A -85,B 0,C 180,E1 -13097.567,E2 -13097.567} C_VEL
LIN {X 0,Y 361.867,Z 263.033,A -85,B 0,C 180,E1 -13100.972,E2 -13100.972} C_VEL
LIN {X 0,Y 361.872,Z 263.012,A -85,B 0,C 180,E1 -13104.654,E2 -13104.654} C_VEL
LIN {X 0,Y 361.835,Z 263.032,A -85,B 0,C 180,E1 -13108.369,E2 -13108.369} C_VEL
LIN {X 0,Y 361.899,Z 263.029,A -85,B 0,C 180,E1 -13110.954,E2 -13110.954} C_VEL
